(* IEC 61131-3 sources: elnaProjects/ElpcLogic/PomarKc7Changed/FunctionBlocks (part 8) *)

(* ---- Pusk_second_faza_chastotny.st ---- *)
FUNCTION_BLOCK Pusk_second_faza_chastotny

VAR_IN_OUT
	StrAlg : struct_Alg;
END_VAR

VAR
	timer120 : struct_PhaseAlgoritm;
	timer5 : struct_PhaseAlgoritm;
	Shup : struct_PhaseAlgoritm;
	Net_Chast : struct_PhaseAlgoritm;
	mvOn : struct_PhaseAlgoritm;
	pGNSmore04 : struct_PhaseAlgoritm;
	gotov_K_zagruzke : struct_PhaseAlgoritm;
	dPmg_Top : struct_PhaseAlgoritm;
	AutoPNS_Start : struct_PhaseAlgoritm;
	fb_timer120 : fb_ph_Timer;
	fb_timer5 : fb_ph_Timer;
	fb_Shup : fb_ph_OilPump;
	fb_Net_Chast : fb_ph_algoritm;
	fb_mvOn : fb_ph_SectionSwitch;
	fb_pGNSmore04 : fb_ph_algoritm;
	fb_gotov_K_zagruzke : fb_ph_algoritm;
	fb_dPmg_Top : fb_ph_algoritm;
	fb_AutoPNS_Start : fb_ph_algoritm;
	_sunpackerCommand : fb_sunpackerCommand;
	_statusDualInput : TYPE_statusDualInput;
	_Answers : TYPE_Answers;
	source : BYTE;
	cmd : BYTE;
	lastCmd : BYTE;
	source_for_Status : BYTE;
	cmd_for_Status : BYTE;
	command_error_for_Status : BYTE;
	resetCmdTimer : TON;
	resetCmdTimerPriznak : BOOL;
	onInit : BOOL;
	waitReset : TON;
END_VAR

VAR_EXTERNAL
	ModeGpa : TYPE_ModeGpa;
	algManager : struct_AlgoritmsManager;
	IM : ImConfig;
	protections : ProtectionsConfig;
	algoritms : AlgoritmsConfig;
	ai : AiConfig;
END_VAR

VAR
	statusAi : TYPE_StatusAi;
END_VAR

IF NOT onInit THEN
         fb_timer120(phaseNumber:=1, delay:=T#120S);
         fb_timer5(phaseNumber:=2, delay:=T#5S);
         fb_Shup(phaseNumber:=3);
         fb_Net_Chast(phaseNumber:=4);
         fb_mvOn(phaseNumber:=5,  act:=_on);
         fb_pGNSmore04(phaseNumber:=6);
         fb_gotov_K_zagruzke(phaseNumber:=7);
         fb_dPmg_Top(phaseNumber:=8);
         fb_AutoPNS_Start(phaseNumber:=9, act:=_run, waitCompletion:=FALSE);
onInit:=TRUE;
END_IF;

fb_timer120(StrPh:=timer120);
fb_timer5(StrPh:= timer5);
fb_Shup(StrPh:= Shup);
fb_Net_Chast(StrPh:=Net_Chast);
fb_mvOn(StrPh:=mvOn, Im:=IM.mv);
fb_pGNSmore04(StrPh:=pGNSmore04);
fb_gotov_K_zagruzke(StrPh:=gotov_K_zagruzke);
fb_dPmg_Top(StrPh:=dPmg_Top);
fb_AutoPNS_Start(StrPh:=AutoPNS_Start, alg:=algoritms.autoPns);

StrAlg.CanRun := StrAlg.inCanRun;
StrAlg.OpcCommandsDisabled := StrAlg.inOpcCommandsDisabled;

IF StrAlg.isRuning THEN
    (* мв не включен - запуск таймера *)
    IF NOT mvOn.top THEN
	runphase(timer120);
    END_IF;
    (* частотный пуск не совершен - запуск таймера *)
    IF NOT Net_Chast.top THEN
	runphase(timer5);
    END_IF;

    (* ШУП не запущен - запуск *)
    IF NOT Shup.start THEN
	runphase(Shup);
    END_IF;

    (* ШУП не завершился - запуск ШУПб МВ *)
    IF NOT Shup.top AND Shup.start THEN
	runIfNotRunningSO(IM.SingleOutputs.Pusk_SHUP);
	Shup.top:=TRUE;
	runphase(mvOn);
    END_IF;

    (* частотный пуск не запущен - запуск *)
    IF NOT Net_Chast.start THEN
	runphase(Net_Chast);
    END_IF;

    (* частотный пуск не завершился - запуск *)
    IF Net_Chast.start AND (NOT Net_Chast.top) THEN
	IF (NOT IM.SingleSignals.Chastotny_pusk.Q) AND (IM.SingleSignals.Chastotny_pusk.status = 1) THEN
		Net_Chast.top:=TRUE;
		resetPhase(timer5);
	END_IF;
    END_IF;

    (* таймер не истек и мв не включен - вовзедение защиты *)
    IF (NOT timer120.top) AND (NOT mvOn.top) THEN
	runDiProtection(protections.Fail_chastotnii_pusk);
    ELSE
	resetDiProtection(protections.Fail_chastotnii_pusk);
    END_IF;

    (* мв не завершился - включение мв *)
    IF mvOn.start AND NOT mvOn.top THEN
	IF IM.mv.onStatus = _statusDualInput.STATUS_ON THEN
              mvOn.top:=TRUE;
	END_IF;
    END_IF;

    (* мв завершился - что-то делаем *)
    IF mvOn.top THEN
	IF NOT pGNSmore04.start (*AND (algManager.mode = ModeGpa.MODE_PUSKPP_Ch OR algManager.mode = ModeGpa.MODE_PUSKAP_Ch)какой режим *) THEN
		runphase(pGNSmore04);
	END_IF;
         (* IF NOT autoAVOM_canrun_flag THEN
              algoritms.AutoAvom.CanRun:=TRUE;
	    autoAVOM_canrun_flag:=TRUE; kto ti
	END_IF;*)
	resetPhase(timer120);
	runphase(gotov_K_zagruzke);

          IF NOT dPmg_Top.start (* AND ((algManager.mode = modegpa.MODE_PUSKAP_Ch) OR (algManager.mode = modegpa.MODE_PUSKPP_Ch))*) THEN
              runphase(dPmg_Top);
	END_IF;

          runAiProtection(protections.Pgaza_na_vyhode_nagnetatelia_GPA_STOP);
	runDiProtection(protections.Off_avar_vikluchatel);
	runDiProtection(protections.Reg_vozb_off);
    END_IF;

    IF dPmg_Top.start AND NOT dPmg_Top.top THEN
	IF NOT IM.SingleSignals.dP_maslo_gaz_Less100.Q AND IM.SingleSignals.dP_maslo_gaz_Less100.status = 1 AND ai.dPmaslo_gaz.value > 150.0 THEN
		dPmg_Top.top:=TRUE;
		runAiProtection(protections.dPmaslo_gaz);
		runDiProtection(protections.dPmaslo_gaz_less100);
		resetAiProtection(protections.Pgaza_na_vhode_nagnetatelia_GPA_STOP);
		resetAiProtection(protections.Pgaza_na_vyhode_nagnetatelia_GPA_STOP);
		algoritms.autoNu.CanRun:=TRUE;
		(*algoritms.autoNu.run(); кого чего, ничего не понимаю *)
	END_IF;
    END_IF;

    IF pGNSmore04.start AND NOT pGNSmore04.top THEN
	IF ai.Pmasla_posle_GNS.interval (*почему интервал, если есть статус *) >= statusAi.NORMAL AND ai.Pmasla_posle_GNS.value > 400.0 THEN
	  	pGNSmore04.top:=TRUE;
	END_IF;
    END_IF;

    IF (pGNSmore04.top AND gotov_K_zagruzke.top AND dPmg_Top.top )(*AND (algManager.mode = modegpa.MODE_PUSKAP_Ch OR (algManager.mode = modegpa.MODE_PUSKPP_Ch) *)OR
	(gotov_K_zagruzke.top) (*AND (algManager.mode = modegpa.MODE_PUSKV_Ch OR algManager.mode = modegpa.MODE_I))*) AND NOT AutoPNS_Start.top  THEN
	algoritms.AutoPns.CanRun :=TRUE;
	(*algoritms.AutoPns;*)
	AutoPNS_Start.top:=TRUE;
    END_IF;

    IF (NOT Net_Chast.top AND timer5.top) OR (timer120.top AND NOT mvOn.top) THEN
	algoritms.ao.CanRun:=TRUE;
	(*algoritms.ao.run ();*)
    END_IF;
END_IF;

StrAlg.CanRun := StrAlg.inCanRun;
StrAlg.OpcCommandsDisabled := StrAlg.inOpcCommandsDisabled;

(* ---- Если управление с ВУ заблокировано, то  передаем команду из алгоритма ---- *)
IF StrAlg.inOpcCommandsDisabled THEN
	StrAlg.inCommand := StrAlg.inCommand_Alg;
ELSE (* иначе передаем команду с АРМа*)
	StrAlg.inCommand := StrAlg.inCommand_ARM;
END_IF;

_sunpackerCommand(command := StrAlg.inCommand);
	source := _sunpackerCommand.source;
	cmd := _sunpackerCommand.cmd;

IF cmd <> 0 AND lastCmd <> cmd AND (((NOT StrAlg.opcCommandsDisabled) AND source > 0) OR source = 0) then
	CASE BYTE_TO_INT(cmd) OF
		(*cmdRun*) 1: 	IF (StrAlg.CanRun) THEN
					StrAlg.isRuning := TRUE;
					StrAlg.isEnded := FALSE;
					StrAlg.hasError := FALSE;
					(*****************       OnRun       *****************)
                                                  algManager.nMode:=ModeGpa.MODE_PUSK_FIRST_FAZA2;

                                                  runPhase(timer120);
                                                  runPhase(timer5);
                                                  runPhase(Shup);
                                                  resetAiProtection(protections.dPmaslo_gaz);
                                                  resetDiProtection(protections.dPmaslo_gaz_less100);

					cmd_for_Status := cmd;
					source_for_Status := source;
					command_error_for_Status := 0;
				ELSE
					StrAlg.isRuning := FALSE;
					StrAlg.isEnded := FALSE;
					StrAlg.hasError := FALSE;

					cmd_for_Status := 0;
					source_for_Status := source;
					command_error_for_Status := cmd;
				END_IF;
		(*cmdReset*) 2: 	StrAlg.isRuning := FALSE;
				StrAlg.isEnded := FALSE;
				StrAlg.hasError 	:= FALSE;

                                         (*****************       OnReset       *****************)
                                        waitReset(IN:=FALSE);
                                        StrAlg.inCanRun:=FALSE;

                                        resetPhase(timer5);
                                        resetPhase(Shup);
                                        resetPhase(timer120);
                                        resetPhase(Net_Chast);
                                        resetPhase(mvOn);
                                        resetPhase(pGNSmore04);
                                        resetPhase(gotov_K_zagruzke);
                                        resetPhase(dPmg_Top);
                                        resetPhase(AutoPNS_Start);

                                        StrAlg.inOpcCommandsDisabled:=FALSE;

				cmd_for_Status := cmd;
				source_for_Status := source;
				command_error_for_Status := 0;
	END_CASE;
	resetCmdTimer(IN := false);
	resetCmdTimerPriznak := TRUE;
END_IF;
lastCmd := cmd;

resetCmdTimer(IN := resetCmdTimerPriznak, PT := T#5S);
IF resetCmdTimer.Q THEN
	resetCmdTimerPriznak := FALSE;
	source_for_Status := 0;
	cmd_for_Status := 0;
	command_error_for_Status := 0;
END_IF;

StrAlg.Start:= timer120.startStatus
            OR timer5.startStatus
            OR Shup.startStatus
            OR Net_Chast.startStatus
            OR mvOn.startStatus
            OR pGNSmore04.startStatus
            OR gotov_K_zagruzke.startStatus
            OR dPmg_Top.startStatus
            OR AutoPNS_Start.startStatus;

StrAlg.Error := timer120.errorStatus
            OR timer5.errorStatus
            OR Shup.errorStatus
            OR Net_Chast.errorStatus
            OR mvOn.errorStatus
            OR pGNSmore04.errorStatus
            OR gotov_K_zagruzke.errorStatus
            OR dPmg_Top.errorStatus
            OR AutoPNS_Start.errorStatus;

StrAlg.Top := timer120.topStatus
            OR timer5.topStatus
            OR Shup.topStatus
            OR Net_Chast.topStatus
            OR mvOn.topStatus
            OR gotov_K_zagruzke.topStatus
            OR dPmg_Top.topStatus
            OR AutoPNS_Start.topStatus
            OR pGNSmore04.topStatus;

(*TODO: TYPE PROGRAM CODE HERE*)
StrAlg.status :=  SHL(BYTE_TO_DWORD(source_for_Status), 29)
			OR SHL(BYTE_TO_DWORD(cmd_for_Status), 26)
			OR SHL(BYTE_TO_DWORD(command_error_for_Status), 23)
			OR SHL(BOOL_TO_DWORD(StrAlg.OpcCommandsDisabled ), 21)
			OR SHL(BOOL_TO_DWORD(StrAlg.hasError),4)
			OR SHL(BOOL_TO_DWORD(StrAlg.CanRun),2)
			OR SHL(BOOL_TO_DWORD(StrAlg.isEnded),1)
			OR BOOL_TO_DWORD(StrAlg.isRuning);

(* ---- Pusk_second_faza_reactor.st ---- *)
FUNCTION_BLOCK Pusk_second_faza_reactor

VAR_IN_OUT
	StrAlg : struct_Alg;
END_VAR

VAR
	timer25 : struct_PhaseAlgoritm;
	timer3 : struct_PhaseAlgoritm;
	mvOn : struct_PhaseAlgoritm;
	pGNSmore04 : struct_PhaseAlgoritm;
	gotov_K_zagruzke : struct_PhaseAlgoritm;
	dPmg_Top : struct_PhaseAlgoritm;
	Mv_Error : struct_PhaseAlgoritm;
	AutoPNS_Start : struct_PhaseAlgoritm;
	fb_timer25 : fb_ph_Timer;
	fb_timer3 : fb_ph_Timer;
	fb_Mv_Error : fb_ph_algoritm;
	fb_mvOn : fb_ph_SectionSwitch;
	fb_pGNSmore04 : fb_ph_algoritm;
	fb_gotov_K_zagruzke : fb_ph_algoritm;
	fb_dPmg_Top : fb_ph_algoritm;
	fb_AutoPNS_Start : fb_ph_algoritm;
	_sunpackerCommand : fb_sunpackerCommand;
	_statusDualInput : TYPE_statusDualInput;
	_Answers : TYPE_Answers;
	source : BYTE;
	cmd : BYTE;
	lastCmd : BYTE;
	source_for_Status : BYTE;
	cmd_for_Status : BYTE;
	command_error_for_Status : BYTE;
	resetCmdTimer : TON;
	resetCmdTimerPriznak : BOOL;
	onInit : BOOL;
	waitReset : TON;
END_VAR

VAR_EXTERNAL
	ModeGpa : TYPE_ModeGpa;
	algManager : struct_AlgoritmsManager;
	IM : ImConfig;
	protections : ProtectionsConfig;
	algoritms : AlgoritmsConfig;
	ai : AiConfig;
END_VAR

VAR
	statusAi : TYPE_StatusAi;
END_VAR

IF NOT onInit THEN
         fb_timer25(phaseNumber:=1, delay:=T#25S);
         fb_timer3(phaseNumber:=2, delay:=T#3S);
         fb_mvOn(phaseNumber:=3, act:=_on);
         fb_pGNSmore04(phaseNumber:=4);
         fb_gotov_K_zagruzke(phaseNumber:=5);
         fb_dPmg_Top(phaseNumber:=6);
         fb_Mv_Error(phaseNumber:=7);
         fb_AutoPNS_start(phaseNumber:=8, act:=_run, waitCompletion:=FALSE);

onInit:=TRUE;
END_IF;

fb_timer25(StrPh:=timer25);
fb_timer3(StrPh:= timer3);
fb_mvOn(StrPh:= mvOn, Im:=IM.mv);
fb_pGNSmore04(StrPh:=pGNSmore04);
fb_gotov_K_zagruzke(StrPh:=gotov_K_zagruzke);
fb_dPmg_Top(StrPh:=dPmg_Top);
fb_Mv_Error(StrPh:=Mv_Error);
fb_AutoPNS_start(StrPh:=AutoPNS_start, alg:=algoritms.autoPns);

StrAlg.CanRun := StrAlg.inCanRun;
StrAlg.OpcCommandsDisabled := StrAlg.inOpcCommandsDisabled;
IF StrAlg.isRuning THEN
    (* если мв не завершен - включаем таймер *)
    IF NOT mvOn.top THEN
        runPhase(timer25);
    END_IF;

    (* если мв не заврешен - включаем таймер *)
    IF NOT mvOn.top THEN
        runPhase(timer3);
    END_IF;

    (* мв не запущен - запускаем мв *)
    IF NOT mvOn.start THEN
        runPhase(mvOn);
    END_IF;

    (* мв завершен *)
    IF mvOn.top  THEN
    (*если проверка пгнс не включена - включаем *)
        IF NOT pGNSmore04.start (*AND ((algManager.mode = modegpa.MODE_PUSKAP_R) OR (algManager.mode = modegpa.MODE_PUSKPP_R))*) THEN
            runPhase(pGNSmore04);
        END_IF;

        (*kakoito flag, hz zachem on
        IF NOT autoAVOM_canrun_flag THEN
            algoritms.S_AutoAVOM.CanRun:=TRUE;
            autoAVOM_canrun_flag:=TRUE;
        END_IF;*)
        resetPhase(timer3);
        resetPhase(timer25);
        Mv_Error.error := FALSE;
        runPhase(gotov_K_zagruzke);
        IF NOT dPmg_Top.start (*AND ((algManager.mode = modegpa.MODE_PUSKAP_R) OR (algManager.mode = modegpa.MODE_PUSKPP_R))*) THEN
            runPhase(dPmg_Top);
        END_IF;

        runDiProtection(protections.mvOff);
        runDiProtection(protections.Off_avar_vikluchatel);
        runDiProtection(protections.Reg_vozb_off);
        ELSIF NOT mvOn.top AND timer3.top THEN
		Mv_Error.error := TRUE;
    END_IF;

    IF	dPmg_Top.start AND NOT dPmg_Top.top THEN
	    IF	NOT IM.SingleSignals.dP_maslo_gaz_Less100.Q AND IM.SingleSignals.dP_maslo_gaz_Less100.status = 1 AND ai.dPmaslo_gaz.value > 150.0	THEN
		    dPmg_Top.top:=TRUE;
		    runAiProtection(protections.dPmaslo_gaz);
		    runDiProtection(protections.dPmaslo_gaz_less100);
		    resetAiProtection(protections.Pgaza_na_vhode_nagnetatelia_GPA_STOP);
		    resetAiProtection(protections.Pgaza_na_vyhode_nagnetatelia_GPA_STOP);
		    (*algoritms.autoNu_2.CanRun:=TRUE;
		    algoritms.autoNu_2.run (); не понимаю*)
	    END_IF;
    END_IF;

    IF	pGNSmore04.start AND NOT pGNSmore04.top THEN
	    IF 	ai.Pmasla_posle_GNS.interval	>=statusAi.NORMAL AND ai.Pmasla_posle_GNS.value	 > 400.0 THEN
	  	    pGNSmore04.top:=TRUE;
	    END_IF;
    END_IF;

    IF	pGNSmore04.top AND gotov_K_zagruzke.top AND dPmg_Top.top (*AND algManager.mode = modegpa.MODE_PUSKAP_R) OR (algManager.mode = modegpa.MODE_PUSKPP_R)))*) OR
	    gotov_K_zagruzke.top (*AND ((algManager.mode = modegpa.MODE_PUSKV_R) OR (algManager.mode = modegpa.MODE_I))))*) AND NOT AutoPNS_start.top  THEN
	    algoritms.AutoPns.CanRun :=TRUE;
	   (*algoritms.AutoPNS_Start.run();*)
	    AutoPNS_start.top:=TRUE;
    END_IF;
    IF	timer25.top AND Mv_Error.error THEN
	algoritms.ao.CanRun:=TRUE;
	(*algoritms.ao.run ();*)
    END_IF;

    (*StrAlg.isEnded:= avom1cmdOff.top AND avom2cmdOff.top;*)
END_IF;
StrAlg.CanRun := StrAlg.inCanRun;
StrAlg.OpcCommandsDisabled := StrAlg.inOpcCommandsDisabled;

(* ---- Если управление с ВУ заблокировано, то  передаем команду из алгоритма ---- *)
IF StrAlg.inOpcCommandsDisabled THEN
	StrAlg.inCommand := StrAlg.inCommand_Alg;
ELSE (* иначе передаем команду с АРМа*)
	StrAlg.inCommand := StrAlg.inCommand_ARM;
END_IF;

_sunpackerCommand(command := StrAlg.inCommand);
	source := _sunpackerCommand.source;
	cmd := _sunpackerCommand.cmd;

IF cmd <> 0 AND lastCmd <> cmd AND (((NOT StrAlg.opcCommandsDisabled) AND source > 0) OR source = 0) then
	CASE BYTE_TO_INT(cmd) OF
		(*cmdRun*) 1: 	IF (StrAlg.CanRun) THEN
					StrAlg.isRuning := TRUE;
					StrAlg.isEnded := FALSE;
					StrAlg.hasError := FALSE;
					(*****************       OnRun       *****************)
                                                  algManager.nMode:=ModeGpa.MODE_PUSK_FIRST_FAZA2;

                                                  (*runPhase(timer120);
                                                  runPhase(timer5);
                                                  runPhase(Shup);
                                                  resetAiProtection(protections.dPmaslo_gaz);
                                                  resetDiProtection(protections.dPmaslo_gaz_less100);*)

					cmd_for_Status := cmd;
					source_for_Status := source;
					command_error_for_Status := 0;
				ELSE
					StrAlg.isRuning := FALSE;
					StrAlg.isEnded := FALSE;
					StrAlg.hasError := FALSE;

					cmd_for_Status := 0;
					source_for_Status := source;
					command_error_for_Status := cmd;
				END_IF;
		(*cmdReset*) 2: 	StrAlg.isRuning := FALSE;
				StrAlg.isEnded := FALSE;
				StrAlg.hasError 	:= FALSE;

                                         (*****************       OnReset       *****************)
                                        waitReset(IN:=FALSE);
                                        StrAlg.inCanRun:=FALSE;

                                        (*resetPhase(timer5);
                                        resetPhase(Shup);
                                        resetPhase(timer120);
                                        resetPhase(Net_Chast);
                                        resetPhase(mvOn);
                                        resetPhase(pGNSmore04);
                                        resetPhase(gotov_K_zagruzke);
                                        resetPhase(dPmg_Top);
                                        resetPhase(AutoPNS_Start);*)

                                        StrAlg.inOpcCommandsDisabled:=FALSE;

				cmd_for_Status := cmd;
				source_for_Status := source;
				command_error_for_Status := 0;
	END_CASE;
	resetCmdTimer(IN := false);
	resetCmdTimerPriznak := TRUE;
END_IF;
lastCmd := cmd;

resetCmdTimer(IN := resetCmdTimerPriznak, PT := T#5S);
IF resetCmdTimer.Q THEN
	resetCmdTimerPriznak := FALSE;
	source_for_Status := 0;
	cmd_for_Status := 0;
	command_error_for_Status := 0;
END_IF;

StrAlg.Start:= timer25.errorStatus
            OR timer3.errorStatus
            OR mvOn.errorStatus
            OR pGNSmore04.errorStatus
            OR gotov_K_zagruzke.errorStatus
            OR dPmg_Top.errorStatus
            OR Mv_Error.errorStatus
            OR AutoPNS_Start.errorStatus;

(*TODO: TYPE PROGRAM CODE HERE*)
StrAlg.status :=  SHL(BYTE_TO_DWORD(source_for_Status), 29)
			OR SHL(BYTE_TO_DWORD(cmd_for_Status), 26)
			OR SHL(BYTE_TO_DWORD(command_error_for_Status), 23)
			OR SHL(BOOL_TO_DWORD(StrAlg.OpcCommandsDisabled ), 21)
			OR SHL(BOOL_TO_DWORD(StrAlg.hasError),4)
			OR SHL(BOOL_TO_DWORD(StrAlg.CanRun),2)
			OR SHL(BOOL_TO_DWORD(StrAlg.isEnded),1)
			OR BOOL_TO_DWORD(StrAlg.isRuning);

(* ---- Pusk_third_faza.st ---- *)
FUNCTION_BLOCK Pusk_third_faza

VAR_IN_OUT
	StrAlg : struct_Alg;
END_VAR

VAR
	timer480 : struct_PhaseAlgoritm;
	kran4Open : struct_PhaseAlgoritm;
	waitAfterKran4 : struct_PhaseAlgoritm;
	kran5Close : struct_PhaseAlgoritm;
	kran3bOpen : struct_PhaseAlgoritm;
	dP_kr1less100 : struct_PhaseAlgoritm;
	Pvh_vyhMore5 : struct_PhaseAlgoritm;
	kran1Open : struct_PhaseAlgoritm;
	kran2Open : struct_PhaseAlgoritm;
	kran3Open : struct_PhaseAlgoritm;
	kran3bClose : struct_PhaseAlgoritm;
	Err_ALG : struct_PhaseAlgoritm;
	fb_timer480 : fb_ph_Timer;
	fb_kran4Open : fb_ph_Kran;
	fb_waitAfterKran4 : fb_ph_Timer;
	fb_kran5Close : fb_ph_Kran;
	fb_kran3bOpen : fb_ph_Kran;
	fb_dP_kr1less100 : fb_ph_algoritm;
	fb_Pvh_vyhMore5 : fb_ph_algoritm;
	fb_kran1Open : fb_ph_Kran;
	fb_kran2Open : fb_ph_Kran;
	fb_kran3Open : fb_ph_Kran;
	fb_kran3bClose : fb_ph_Kran;
	fb_Err_ALG : fb_ph_algoritm;
	_sunpackerCommand : fb_sunpackerCommand;
	_statusDualInput : TYPE_statusDualInput;
	_Answers : TYPE_Answers;
	source : BYTE;
	cmd : BYTE;
	lastCmd : BYTE;
	source_for_Status : BYTE;
	cmd_for_Status : BYTE;
	command_error_for_Status : BYTE;
	resetCmdTimer : TON;
	resetCmdTimerPriznak : BOOL;
	onInit : BOOL;
	waitReset : TON;
END_VAR

VAR_EXTERNAL
	ModeGpa : TYPE_ModeGpa;
	algManager : struct_AlgoritmsManager;
	IM : ImConfig;
	protections : ProtectionsConfig;
	algoritms : AlgoritmsConfig;
	ai : AiConfig;
END_VAR

VAR
	statusAi : TYPE_StatusAi;
END_VAR

IF NOT onInit THEN
         fb_timer480(phaseNumber:=1, delay:=T#480S);
         fb_kran4Open(phaseNumber:=2, act:=_on);
         fb_waitAfterKran4(phaseNumber:=3, delay:=T#10S);
         fb_kran5Close(phaseNumber:=4, act:=_off);
         fb_kran3bOpen(phaseNumber:=5, act:=_on);
         fb_dP_kr1less100(phaseNumber:=6);
         fb_Pvh_vyhMore5(phaseNumber:=7);
         fb_kran1Open(phaseNumber:=8, act:=_on);
         fb_kran2Open(phaseNumber:=9, act:=_on);
         fb_kran3Open(phaseNumber:=10, act:=_on);
         fb_kran3bClose(phaseNumber:=11, act:=_off);
         fb_Err_ALG(phaseNumber:=12);
onInit:=TRUE;
END_IF;

fb_timer480(StrPh:=timer480);
fb_kran4Open(StrPh:= kran4Open, Im:=Im.kran4);
fb_waitAfterKran4(StrPh:= waitAfterKran4);
fb_kran5Close(StrPh:=kran5Close, Im:=Im.kran5);
fb_kran3bOpen(StrPh:=kran3bOpen, Im:=Im.kran3b);
fb_dP_kr1less100(StrPh:=dP_kr1less100);
fb_Pvh_vyhMore5(StrPh:=Pvh_vyhMore5);
fb_kran1Open(StrPh:=kran1Open, Im:=Im.kran1);
fb_kran2Open(StrPh:=kran2Open, Im:=Im.kran2);
fb_kran3Open(StrPh:=kran3Open, Im:=Im.kran3);
fb_kran3bClose(StrPh:=kran3bClose, Im:=Im.kran3b);
fb_Err_ALG(StrPh:=Err_ALG);

StrAlg.CanRun := StrAlg.inCanRun;
StrAlg.OpcCommandsDisabled := StrAlg.inOpcCommandsDisabled;

IF StrAlg.isRuning THEN
    (* запуск таймера *)
    IF NOT (kran3bClose.top) THEN
	    runPhase(timer480);
    END_IF;

    (*если кран1 не открыт - октрыть кран 4*)
    IF	NOT kran1Open.top (*AND IM.kran4._cmdreset.IN = FALSE*)  THEN
	    runIfNotRunningSO(IM.SingleOutputs.Kr4_open_from_alg);
	    runPhase(kran4Open);
    END_IF;
    IF	kran4Open.start AND NOT kran4Open.top THEN
	    IF	IM.kran4.onStatus = _statusDualInput.STATUS_ON THEN
		    kran4Open.top:=TRUE;
	    END_IF;
    END_IF;

    (* продувка крана *)
    IF kran4Open.top THEN
        runPhase(waitAfterKran4);
    END_IF;

    (* кран продулся - закрытие кран 5*)
    IF waitAfterKran4.top THEN
	    runPhase(kran5Close);
    END_IF;

    (* кран 5 закрыт - открытие крана 3б проверка перепада давление*)
    IF	kran5Close.top THEN
	    runPhase(kran3bOpen);
	    runPhase(dP_kr1less100);
	    runPhase(Pvh_vyhMore5);
    END_IF;

    (* проверка давления крана *)
    IF	Pvh_vyhMore5.start AND NOT Pvh_vyhMore5.top THEN
	    IF	(ai.Pgaza_na_vhode_nagnetatelia.interval >=statusAi.NORMAL) AND (ai.Pgaza_na_vhode_nagnetatelia.value	 >= 4.0) AND
		    (ai.Pgaza_na_vyhode_nagnetatelia.interval >=statusAi.NORMAL) AND (ai.Pgaza_na_vyhode_nagnetatelia.value	 >= 4.0) THEN
		        Pvh_vyhMore5.top := TRUE;
    		    runAiProtection(protections.Pgaza_na_vyhode_nagnetatelia);
	    END_IF;
    END_IF;

    (* проверка открытия крана 3б *)
    IF	kran3bOpen.start AND NOT kran3bOpen.top THEN
	    IF	IM.kran3b.onStatus=_statusDualInput.STATUS_ON THEN
		    kran3bOpen.top :=TRUE;
	    END_IF;
    END_IF;
    IF	kran3bOpen.top AND	kran5Close.top AND dP_kr1less100.top AND Pvh_vyhMore5.top THEN
	    runPhase(kran1Open);
	    runPhase(kran2Open);
	    runPhase(kran3Open);
	    (*Smazka_1_2:=TRUE; нет такого *)
    END_IF;
    IF	kran1Open.top THEN
	    resetIfRunningSO(IM.SingleOutputs.Kr4_open_from_alg);
	    (*ystavki.Block_kr4_alg.setValue (0);что такое уставки*)
    END_IF;

    (* закрытие крана 3бис *)
    IF kran1Open.top AND kran2Open.top AND kran3Open.top THEN
	    runPhase(kran3bClose);
    END_IF;
    IF 	kran3bClose.top THEN
	    Err_ALG.error :=FALSE;
	    resetPhase(timer480);
    ELSIF NOT kran3bClose.top AND timer480.top THEN
		Err_ALG.error :=TRUE;
    END_IF;
END_IF;

_sunpackerCommand(command := StrAlg.inCommand);
	source := _sunpackerCommand.source;
	cmd := _sunpackerCommand.cmd;

IF cmd <> 0 AND lastCmd <> cmd AND (((NOT StrAlg.opcCommandsDisabled) AND source > 0) OR source = 0) then
	CASE BYTE_TO_INT(cmd) OF
		(*cmdRun*) 1: 	IF (StrAlg.CanRun) THEN
					StrAlg.isRuning := TRUE;
					StrAlg.isEnded := FALSE;
					StrAlg.hasError := FALSE;
					(*****************       OnRun       *****************)
                                                  algManager.nMode:=ModeGpa.MODE_PUSK_FIRST_FAZA2;

                                                  (*runPhase(timer120);
                                                  runPhase(timer5);
                                                  runPhase(Shup);
                                                  resetAiProtection(protections.dPmaslo_gaz);
                                                  resetDiProtection(protections.dPmaslo_gaz_less100);*)

					cmd_for_Status := cmd;
					source_for_Status := source;
					command_error_for_Status := 0;
				ELSE
					StrAlg.isRuning := FALSE;
					StrAlg.isEnded := FALSE;
					StrAlg.hasError := FALSE;

					cmd_for_Status := 0;
					source_for_Status := source;
					command_error_for_Status := cmd;
				END_IF;
		(*cmdReset*) 2: 	StrAlg.isRuning := FALSE;
				StrAlg.isEnded := FALSE;
				StrAlg.hasError 	:= FALSE;

                                         (*****************       OnReset       *****************)
                                        waitReset(IN:=FALSE);
                                        StrAlg.inCanRun:=FALSE;

                                        (*resetPhase(timer5);
                                        resetPhase(Shup);
                                        resetPhase(timer120);
                                        resetPhase(Net_Chast);
                                        resetPhase(mvOn);
                                        resetPhase(pGNSmore04);
                                        resetPhase(gotov_K_zagruzke);
                                        resetPhase(dPmg_Top);
                                        resetPhase(AutoPNS_Start);*)

                                        StrAlg.inOpcCommandsDisabled:=FALSE;

				cmd_for_Status := cmd;
				source_for_Status := source;
				command_error_for_Status := 0;
	END_CASE;
	resetCmdTimer(IN := false);
	resetCmdTimerPriznak := TRUE;
END_IF;
lastCmd := cmd;

resetCmdTimer(IN := resetCmdTimerPriznak, PT := T#5S);
IF resetCmdTimer.Q THEN
	resetCmdTimerPriznak := FALSE;
	source_for_Status := 0;
	cmd_for_Status := 0;
	command_error_for_Status := 0;
END_IF;

StrAlg.Start:= timer480.startStatus
            OR kran4Open.startStatus
            OR waitAfterKran4.startStatus
            OR kran5Close.startStatus
            OR kran3bOpen.startStatus
            OR dP_kr1less100.startStatus
            OR Pvh_vyhMore5.startStatus
            OR kran1Open.startStatus
            OR kran2Open.startStatus
            OR kran3Open.startStatus
            OR kran3bClose.startStatus
            OR Err_ALG.startStatus;

StrAlg.Error := timer480.errorStatus
            OR kran4Open.errorStatus
            OR waitAfterKran4.errorStatus
            OR kran5Close.errorStatus
            OR kran3bOpen.errorStatus
            OR dP_kr1less100.errorStatus
            OR Pvh_vyhMore5.errorStatus
            OR kran1Open.errorStatus
            OR kran2Open.errorStatus
            OR kran3Open.errorStatus
            OR kran3bClose.errorStatus
            OR Err_ALG.errorStatus;

StrAlg.Top := timer480.topStatus
            OR kran4Open.topStatus
            OR waitAfterKran4.topStatus
            OR kran5Close.topStatus
            OR kran3bOpen.topStatus
            OR dP_kr1less100.topStatus
            OR Pvh_vyhMore5.topStatus
            OR kran1Open.topStatus
            OR kran2Open.topStatus
            OR kran3Open.topStatus
            OR kran3bClose.topStatus
            OR Err_ALG.topStatus;

(*TODO: TYPE PROGRAM CODE HERE*)
StrAlg.status :=  SHL(BYTE_TO_DWORD(source_for_Status), 29)
			OR SHL(BYTE_TO_DWORD(cmd_for_Status), 26)
			OR SHL(BYTE_TO_DWORD(command_error_for_Status), 23)
			OR SHL(BOOL_TO_DWORD(StrAlg.OpcCommandsDisabled ), 21)
			OR SHL(BOOL_TO_DWORD(StrAlg.hasError),4)
			OR SHL(BOOL_TO_DWORD(StrAlg.CanRun),2)
			OR SHL(BOOL_TO_DWORD(StrAlg.isEnded),1)
			OR BOOL_TO_DWORD(StrAlg.isRuning);

(* ---- puskKalg.st ---- *)
FUNCTION_BLOCK puskKalg

VAR_IN_OUT
	StrAlg : struct_Alg;
END_VAR

VAR
	puskOilSystem : struct_PhaseAlgoritm;
END_VAR

VAR_IN_OUT
	questionFilling : struct_Question;
END_VAR

VAR
	filling : struct_PhaseAlgoritm;
END_VAR

VAR_IN_OUT
	questionUnload : struct_Question;
END_VAR

VAR
	kran3bOpen : struct_PhaseAlgoritm;
	kran4Close : struct_PhaseAlgoritm;
	kran1Close : struct_PhaseAlgoritm;
	kran2Close : struct_PhaseAlgoritm;
	kran5open : struct_PhaseAlgoritm;
	wait720 : struct_PhaseAlgoritm;
	noGasInPipe : struct_PhaseAlgoritm;
	AutoNUoff : struct_PhaseAlgoritm;
	nu1Off : struct_PhaseAlgoritm;
	nu2Off : struct_PhaseAlgoritm;
	pnsWaitOff : struct_PhaseAlgoritm;
	testUnsuccessfulUnfill : struct_PhaseAlgoritm;
	fb_puskOilSystem : fb_ph_algoritm;
	fb_questionFilling : fb_Question;
	fb_filling : fb_ph_algoritm;
	fb_questionUnload : fb_Question;
	fb_kran3bOpen : fb_ph_Kran;
	fb_kran4Close : fb_ph_CustomPhase;
	fb_kran1Close : fb_ph_Kran;
	fb_kran2Close : fb_ph_Kran;
	fb_kran5open : fb_ph_Kran;
	fb_wait720 : fb_ph_Timer;
	fb_noGasInPipe : fb_ph_CustomPhase;
	fb_AutoNUoff : fb_ph_algoritm;
	fb_nu1Off : fb_ph_OilPump;
	fb_nu2Off : fb_ph_OilPump;
	fb_pnsWaitOff : fb_ph_algoritm;
	fb_testUnsuccessfulUnfill : fb_ph_CustomPhase;
	_sunpackerCommand : fb_sunpackerCommand;
	_DualStateImAction : TYPE_DualStateImAction;
	_Answers : TYPE_Answers;
	_statusDualInput : TYPE_statusDualInput;
	_StatusAi : TYPE_StatusAi;
	_PhaseAlgoritmAction : TYPE_PhaseAlgoritmAction;
	source : BYTE;
	cmd : BYTE;
	lastCmd : BYTE;
	source_for_Status : BYTE;
	cmd_for_Status : BYTE;
	command_error_for_Status : BYTE;
	resetCmdTimer : TON;
	resetCmdTimerPriznak : BOOL;
	OpcCommandsKransEnabled : BOOL;
	OpcCommandsKransDisabled : BOOL;
	_resetQuestion1 : BOOL;
	_resetQuestion2 : BOOL;
	onInit : BOOL;
	waitReset : TON;
END_VAR

VAR_EXTERNAL
	IM : ImConfig;
	algoritms : AlgoritmsConfig;
	ai : AiConfig;
	AlgTimers : struct_AlgTimers;
	ModeGpa : TYPE_ModeGpa;
	algManager : struct_AlgoritmsManager;
	protections : ProtectionsConfig;
END_VAR

VAR CONSTANT
	Ust_Pgaza : LREAL          := 0.3;
END_VAR

IF NOT onInit THEN

          fb_puskOilSystem(phaseNumber:=0, act:=_run, waitCompletion:=TRUE);
      questionFilling.AnswerVariants:=_Answers.ANS_YES;
                fb_filling(phaseNumber:=1, act:=_run, waitCompletion:=TRUE);
    questionUnload.AnswerVariants:=_Answers.ANS_YES;
             fb_kran3bOpen(phaseNumber:=3, act:=_on);
             fb_kran4Close(phaseNumber:=4);
             fb_kran1Close(phaseNumber:=5, act:=_off);
             fb_kran2Close(phaseNumber:=6, act:=_off);
              fb_kran5open(phaseNumber:=7, act:=_on);
                fb_wait720(phaseNumber:=8, delay:=T#720S);
            fb_noGasInPipe(phaseNumber:=9);
              fb_AutoNUoff(phaseNumber:=10, act:=_reset, waitCompletion:=FALSE);
                 fb_nu1Off(phaseNumber:=11, act:=_off);
                 fb_nu2Off(phaseNumber:=12, act:=_off);
             fb_pnsWaitOff(phaseNumber:=15, act:=_run, waitCompletion:=TRUE);
 fb_testUnsuccessfulUnfill(phaseNumber:=18);

onInit:=TRUE;
END_IF;

          fb_puskOilSystem(StrPh:=puskOilSystem, alg:=algoritms.puskOilSystem);
        fb_questionFilling(StrQ:=questionFilling);
                fb_filling(StrPh:=filling, alg:=algoritms.filling);
         fb_questionUnload(StrQ:=questionUnload);
             fb_kran3bOpen(StrPh:=kran3bOpen, Im:=Im.kran3b);
             fb_kran4Close(StrPh:=kran4Close);
             fb_kran1Close(StrPh:=kran1Close, Im:=Im.kran1);
             fb_kran2Close(StrPh:=kran2Close, Im:=Im.kran2);
              fb_kran5open(StrPh:=kran5open, Im:=Im.kran5);
                fb_wait720(StrPh:=wait720, timer:=AlgTimers.puskK_wait720);
            fb_noGasInPipe(StrPh:=noGasInPipe);
              fb_AutoNUoff(StrPh:=AutoNUoff, alg:=algoritms.autoNu);
                 fb_nu1Off(StrPh:=nu1Off, Im:=Im.nu1);
                 fb_nu2Off(StrPh:=nu2Off, Im:=Im.nu2);
             fb_pnsWaitOff(StrPh:=pnsWaitOff, alg:=algoritms.vibegPNS);
 fb_testUnsuccessfulUnfill(StrPh:=testUnsuccessfulUnfill);

StrAlg.CanRun := StrAlg.inCanRun;
StrAlg.OpcCommandsDisabled := StrAlg.inOpcCommandsDisabled;

IF StrAlg.isRuning THEN

    StrAlg.hasError := kran3bOpen.error OR kran1Close.error OR kran2Close.error OR kran5open.error OR testUnsuccessfulUnfill.error;

    IF puskOilSystem.top THEN
         IF NOT _resetQuestion1 THEN
         askQuestion(questionFilling);
         _resetQuestion1:=TRUE;
         END_IF;
    END_IF;

    IF questionFilling.answer = _Answers.ANS_YES THEN
        runPhase(filling);
        resetQuestion(questionFilling);
    END_IF;

    IF filling.top THEN
       OpcCommandsKransEnabled:=TRUE;
       resetDiProtection(protections.Reg_vozb_off);
       (*resetDiProtection(protections.Fail_chastotnii_pusk);*)
       IF NOT _resetQuestion2 THEN
       askQuestion(questionUnload);
       _resetQuestion2:=TRUE;
       END_IF;
    END_IF;

     IF questionUnload.answer = _Answers.ANS_YES THEN
        OpcCommandsKransDisabled:=TRUE;
        runPhase(kran3bOpen);
        runPhase(wait720);
        resetQuestion(questionUnload);
    END_IF;

    IF kran3bOpen.top THEN
          resetDiProtection(protections.Reg_vozb_off);
          resetDiProtection(protections.Fail_chastotnii_pusk);

          runPhase(kran1Close);
          runPhase(kran2Close);
          runPhase(kran4Close);
    END_IF;

     IF kran4Close.start AND NOT kran4Close.top THEN
	kran4Close.top:= Im.kran4.onStatus = _statusDualInput.STATUS_OFF;
    END_IF;

    IF kran1Close.top AND kran2Close.top AND kran4Close.top THEN
	runPhase(kran5open);
    END_IF;

    IF kran5open.top THEN
	runPhase(noGasInPipe);
    END_IF;

    IF noGasInPipe.start AND (NOT noGasInPipe.top) THEN
	noGasInPipe.top:=  (ai.dPgaza_na_maslo_filtre.interval >= _statusAi.NORMAL
                         AND  ai.dPgaza_na_maslo_filtre.value< Ust_Pgaza )
                         AND (ai.Pmaslo_sm_vysokoe.interval >= _statusAi.NORMAL
                         AND  ai.Pmaslo_sm_vysokoe.value< Ust_Pgaza);
    END_IF;

    IF noGasInPipe.top THEN

          ai.Tmasla_MB.Disabled_LA:=TRUE;
          ai.Tmasla_MB.Disabled_LW:=TRUE;
          (*IM.SingleSignals.dP_oilgaz_low.Disabled_Sig:=TRUE;*)
          resetAiProtection(protections.Os_sdvig_nagnetatelja_plus);
         (* resetDiProtection(protections.Vibro_skorost_OP_shesterni_RED_T5);*)
	runPhase(AutoNUoff);

    END_IF;

     IF autoNuOff.top THEN
	runPhase(nu1off);
          runPhase(nu2off);
    END_IF;

    IF nu1Off.top AND nu2Off.top THEN
	runPhase(pnsWaitOff);
    END_IF;

    IF wait720.top AND NOT (pnsWaitOff.top) THEN
          testUnsuccessfulUnfill.error:=TRUE;
    END_IF;

    IF pnsWaitOff.top THEN
          resetPhase(wait720);
	waitReset(IN:=TRUE, PT:= T#3S);
    END_IF;

    IF waitReset.Q THEN
        resetIfRunning(algoritms.vibegPNS);
        algManager.nMode:=ModeGpa.MODE_STOP;
        resetIfRunning(StrAlg);
    END_IF;

    StrAlg.isEnded:= pnsWaitOff.top;

    IF OpcCommandsKransEnabled AND NOT OpcCommandsKransDisabled THEN
	IF      (im.pns.onStatus = _statusDualInput.STATUS_ON)
              AND (im.nu1.onStatus = _statusDualInput.STATUS_ON OR im.nu2.onStatus = _statusDualInput.STATUS_ON)
	    AND (ai.Tmasla_MB.interval >= _statusAi.normal)
              (*AND (ai.Tmasla_MB.value > im.PuskOilSystem_UstdPmg.Value)*)
          THEN
	    IM.Kran3b.inOpcCommandsDisabled:=FALSE;
	    Im.kran4.inOpcCommandsDisabled:=FALSE;
	    Im.kran5.inOpcCommandsDisabled:=FALSE;
		(*IF	Im.SingleSignals.dP_gazgaz_Kran1.q THEN
			Im.kran1.inOpcCommandsDisabled:=FALSE;
			Im.kran2.inOpcCommandsDisabled:=FALSE;
		ELSE
			Im.kran1.inOpcCommandsDisabled:=TRUE;
			Im.kran2.inOpcCommandsDisabled:=TRUE;
		END_IF;*)
          ELSE
	    Im.kran1.inOpcCommandsDisabled:=TRUE;
	    Im.kran2.inOpcCommandsDisabled:=TRUE;
	    Im.kran3b.inOpcCommandsDisabled:=TRUE;
	    Im.kran4.inOpcCommandsDisabled:=TRUE;
	    Im.kran5.inOpcCommandsDisabled:=TRUE;
          END_IF;

    ELSE
	Im.kran1.inOpcCommandsDisabled:=TRUE;
	Im.kran2.inOpcCommandsDisabled:=TRUE;
	Im.kran3b.inOpcCommandsDisabled:=TRUE;
	Im.kran4.inOpcCommandsDisabled:=TRUE;
	Im.kran5.inOpcCommandsDisabled:=TRUE;
    END_IF;
END_IF;

StrAlg.CanRun := StrAlg.inCanRun;
StrAlg.OpcCommandsDisabled := StrAlg.inOpcCommandsDisabled;

(* ---- Если управление с ВУ заблокировано, то  передаем команду из алгоритма ---- *)
IF StrAlg.inOpcCommandsDisabled THEN
	StrAlg.inCommand := StrAlg.inCommand_Alg;
ELSE (* иначе передаем команду с АРМа*)
	StrAlg.inCommand := StrAlg.inCommand_ARM;
END_IF;

_sunpackerCommand(command := StrAlg.inCommand);
	source := _sunpackerCommand.source;
	cmd := _sunpackerCommand.cmd;

IF cmd <> 0 AND lastCmd <> cmd AND (((NOT StrAlg.opcCommandsDisabled) AND source > 0) OR source = 0) then
	CASE BYTE_TO_INT(cmd) OF
		(*cmdRun*) 1: 	IF (StrAlg.CanRun) THEN
					StrAlg.isRuning := TRUE;
					StrAlg.isEnded := FALSE;
					StrAlg.hasError := FALSE;
					(*****************       OnRun       *****************)

                                                  algManager.nMode:=ModeGpa.MODE_PUSKK;
                                                  resetAndDisable(alg:=algoritms.ppu);
                                                  algoritms.puskOilSystem.inCanRun:= TRUE;
                                                  algoritms.filling.inCanRun:= TRUE;
                                                  runPhase(puskOilSystem);

					cmd_for_Status := cmd;
					source_for_Status := source;
					command_error_for_Status := 0;
				ELSE
					StrAlg.isRuning := FALSE;
					StrAlg.isEnded := FALSE;
					StrAlg.hasError 	:= FALSE;

					cmd_for_Status := 0;
					source_for_Status := source;
					command_error_for_Status := cmd;
				END_IF;
		(*cmdReset*) 2: 	StrAlg.isRuning := FALSE;
				StrAlg.isEnded := FALSE;
				StrAlg.hasError 	:= FALSE;

                                         (*****************       OnReset       *****************)
                                        OpcCommandsKransEnabled:=FALSE;
                                        OpcCommandsKransDisabled:=FALSE;
                                        waitReset(IN:=FALSE);
                                        _resetQuestion1:=FALSE;
                                        _resetQuestion2:=FALSE;
                                        resetPhase(puskOilSystem);
                                        resetPhase(filling);
                                        resetPhase(kran3bOpen);
                                        resetPhase(kran4Close);
                                        resetPhase(kran1Close);
                                        resetPhase(kran2Close);
                                        resetPhase(kran5open);
                                        resetPhase(wait720);
                                        resetPhase(noGasInPipe);
                                        resetPhase(AutoNUoff);
                                        resetPhase(nu1Off);
                                        resetPhase(nu2Off);
                                        resetPhase(pnsWaitOff);
                                        resetPhase(testUnsuccessfulUnfill);
                                        BlockAllIM(IM);
                                        resetQuestion(questionFilling);
                                        resetQuestion(questionUnload);

                                        StrAlg.inOpcCommandsDisabled:=FALSE;

				cmd_for_Status := cmd;
				source_for_Status := source;
				command_error_for_Status := 0;
	END_CASE;
	resetCmdTimer(IN := false);
	resetCmdTimerPriznak := TRUE;
END_IF;
lastCmd := cmd;

resetCmdTimer(IN := resetCmdTimerPriznak, PT := T#5S);
IF resetCmdTimer.Q THEN
	resetCmdTimerPriznak := FALSE;
	source_for_Status := 0;
	cmd_for_Status := 0;
	command_error_for_Status := 0;
END_IF;

StrAlg.Start:= puskOilSystem.startStatus
            OR filling.startStatus
            OR kran3bOpen.startStatus
            OR kran4Close.startStatus
            OR kran1Close.startStatus
            OR kran2Close.startStatus
            OR kran5open.startStatus
            OR wait720.startStatus
            OR noGasInPipe.startStatus
            OR AutoNUoff.startStatus
            OR nu1Off.startStatus
            OR nu2Off.startStatus
            OR pnsWaitOff.startStatus
            OR testUnsuccessfulUnfill.startStatus;

StrAlg.Error:=  puskOilSystem.errorStatus
            OR filling.errorStatus
            OR kran3bOpen.errorStatus
            OR kran4Close.errorStatus
            OR kran1Close.errorStatus
            OR kran2Close.errorStatus
            OR kran5open.errorStatus
            OR wait720.errorStatus
            OR noGasInPipe.errorStatus
            OR AutoNUoff.errorStatus
            OR nu1Off.errorStatus
            OR nu2Off.errorStatus
            OR pnsWaitOff.errorStatus
            OR testUnsuccessfulUnfill.errorStatus;

StrAlg.Top:=   puskOilSystem.topStatus
            OR filling.topStatus
            OR kran3bOpen.topStatus
            OR kran4Close.topStatus
            OR kran1Close.topStatus
            OR kran2Close.topStatus
            OR kran5open.topStatus
            OR wait720.topStatus
            OR noGasInPipe.topStatus
            OR AutoNUoff.topStatus
            OR nu1Off.topStatus
            OR nu2Off.topStatus
            OR pnsWaitOff.topStatus
            OR testUnsuccessfulUnfill.topStatus;

(*TODO: TYPE PROGRAM CODE HERE*)
StrAlg.status :=  SHL(BYTE_TO_DWORD(source_for_Status), 29)
			OR SHL(BYTE_TO_DWORD(cmd_for_Status), 26)
			OR SHL(BYTE_TO_DWORD(command_error_for_Status), 23)
			OR SHL(BOOL_TO_DWORD(StrAlg.OpcCommandsDisabled ), 21)
			OR SHL(BOOL_TO_DWORD(StrAlg.hasError),4)
			OR SHL(BOOL_TO_DWORD(StrAlg.CanRun),2)
			OR SHL(BOOL_TO_DWORD(StrAlg.isEnded),1)
			OR BOOL_TO_DWORD(StrAlg.isRuning);

(* ---- puskValg.st ---- *)
FUNCTION_BLOCK puskValg

VAR_IN_OUT
	StrAlg : struct_Alg;
END_VAR

VAR
	puskOilSystem : struct_PhaseAlgoritm;
END_VAR

VAR_IN_OUT
	questionEngine : struct_Question;
END_VAR

VAR
	runningEngine : struct_PhaseAlgoritm;
END_VAR

VAR_IN_OUT
	questionMVoff : struct_Question;
END_VAR

VAR
	mvOff : struct_PhaseAlgoritm;
	pnsOn : struct_PhaseAlgoritm;
	wait600 : struct_PhaseAlgoritm;
	AutoNUoff : struct_PhaseAlgoritm;
	nu1Off : struct_PhaseAlgoritm;
	nu2Off : struct_PhaseAlgoritm;
	autoAvomOff : struct_PhaseAlgoritm;
	Avom1Off : struct_PhaseAlgoritm;
	Avom2Off : struct_PhaseAlgoritm;
	pnsWaitOff : struct_PhaseAlgoritm;
	testUnsuccessful : struct_PhaseAlgoritm;
	fb_puskOilSystem : fb_ph_algoritm;
	fb_questionEngine : fb_Question;
	fb_runningEngine : fb_ph_algoritm;
	fb_questionMVoff : fb_Question;
	fb_mvOff : fb_ph_SectionSwitch;
	fb_pnsOn : fb_ph_Switch;
	fb_wait600 : fb_ph_Timer;
	fb_AutoNUoff : fb_ph_algoritm;
	fb_nu1Off : fb_ph_OilPump;
	fb_nu2Off : fb_ph_OilPump;
	fb_autoAvomOff : fb_ph_algoritm;
	fb_Avom1Off : fb_ph_Switch;
	fb_Avom2Off : fb_ph_Switch;
	fb_pnsWaitOff : fb_ph_algoritm;
	fb_testUnsuccessful : fb_ph_CustomPhase;
	_sunpackerCommand : fb_sunpackerCommand;
	_DualStateImAction : TYPE_DualStateImAction;
	_Answers : TYPE_Answers;
	_statusDualInput : TYPE_statusDualInput;
	_StatusAi : TYPE_StatusAi;
	_PhaseAlgoritmAction : TYPE_PhaseAlgoritmAction;
	source : BYTE;
	cmd : BYTE;
	lastCmd : BYTE;
	source_for_Status : BYTE;
	cmd_for_Status : BYTE;
	command_error_for_Status : BYTE;
	resetCmdTimer : TON;
	resetCmdTimerPriznak : BOOL;
	onInit : BOOL;
	_resetQuestion1 : BOOL;
	_resetQuestion2 : BOOL;
	waitReset : TON;
END_VAR

VAR_EXTERNAL
	IM : ImConfig;
	algoritms : AlgoritmsConfig;
	ai : AiConfig;
	AlgTimers : struct_AlgTimers;
	ModeGpa : TYPE_ModeGpa;
	algManager : struct_AlgoritmsManager;
	protections : ProtectionsConfig;
END_VAR

VAR CONSTANT
	Ust_Pgaza : LREAL          := 0.3;
END_VAR

IF NOT onInit THEN

          fb_puskOilSystem(phaseNumber:=0, act:=_run, waitCompletion:=TRUE);
       questionEngine.AnswerVariants:=_Answers.ANS_YES;
          fb_runningEngine(phaseNumber:=1, act:=_run, waitCompletion:=TRUE);
        questionMVoff.AnswerVariants:=_Answers.ANS_YES;
                  fb_mvOff(phaseNumber:=3, act:=_off);
                  fb_pnsOn(phaseNumber:=4, act:=_on);
                fb_wait600(phaseNumber:=8, delay:=T#600S);
              fb_AutoNUoff(phaseNumber:=10, act:=_reset, waitCompletion:=FALSE);
                 fb_nu1Off(phaseNumber:=11, act:=_off);
                 fb_nu2Off(phaseNumber:=12, act:=_off);
             fb_pnsWaitOff(phaseNumber:=15, act:=_run, waitCompletion:=TRUE);
            fb_autoAvomOff(phaseNumber:=7, act:=_reset, waitCompletion:=FALSE);
               fb_Avom1Off(phaseNumber:=5, act:=_off);
               fb_Avom2Off(phaseNumber:=6, act:=_off);
       fb_testUnsuccessful(phaseNumber:=17);

onInit:=TRUE;
END_IF;

          fb_puskOilSystem(StrPh:=puskOilSystem, alg:=algoritms.puskOilSystem);
         fb_questionEngine(StrQ:=questionEngine);
          fb_runningEngine(StrPh:=runningEngine, alg:=algoritms.engineRun);
          fb_questionMVoff(StrQ:=questionMVoff);
                  fb_mvOff(StrPh:=mvOff, Im:=Im.mv);
                  fb_pnsOn(StrPh:=pnsOn, Im:=Im.pns);
                fb_wait600(StrPh:=wait600, timer:=AlgTimers.puskV_wait600);
              fb_AutoNUoff(StrPh:=AutoNUoff, alg:=algoritms.autoNu);
                 fb_nu1Off(StrPh:=nu1Off, Im:=Im.nu1);
                 fb_nu2Off(StrPh:=nu2Off, Im:=Im.nu2);
             fb_pnsWaitOff(StrPh:=pnsWaitOff, alg:=algoritms.vibegPNS);
            fb_autoAvomOff(StrPh:=autoAvomOff, alg:=algoritms.AutoAvom);
               fb_Avom1Off(StrPh:=Avom1Off, Im:=Im.v1_Avom);
               fb_Avom2Off(StrPh:=Avom2Off, Im:=Im.v2_Avom);
       fb_testUnsuccessful(StrPh:=testUnsuccessful);

StrAlg.CanRun := StrAlg.inCanRun;
StrAlg.OpcCommandsDisabled := StrAlg.inOpcCommandsDisabled;

IF StrAlg.isRuning THEN

    StrAlg.hasError := mvOff.error OR pnsOn.error OR testUnsuccessful.error;

    IF puskOilSystem.top THEN
         IF NOT _resetQuestion1 THEN
         askQuestion(questionEngine);
         _resetQuestion1:=TRUE;
         END_IF;
    END_IF;

    IF questionEngine.answer = _Answers.ANS_YES THEN
        runPhase(runningEngine);
        resetQuestion(questionEngine);
    END_IF;

    IF runningEngine.top THEN
       IF NOT _resetQuestion2 THEN
       askQuestion(questionMVoff);
       _resetQuestion2:=TRUE;
       END_IF;
    END_IF;

     IF questionMVoff.answer = _Answers.ANS_YES THEN

        (*resetDiProtection(protections.Pgaza_na_vyhode_nagnetatelia_GPA_STOP);
       *) resetIfRunning(algoritms.AutoPns);
        runPhase(mvOff);
        runPhase(wait600);
        resetQuestion(questionMVoff);
     END_IF;

    IF mvOff.top THEN
        runPhase(pnsOn);
    END_IF;

    IF pnsOn.top THEN

          ai.Tmasla_MB.Disabled_LA:=TRUE;
          ai.Tmasla_MB.Disabled_LW:=TRUE;
          (*IM.SingleSignals.dP_oilgaz_low.Disabled_Sig:=TRUE;*)
          (*resetAiProtection(protections.Os_sdvig_nagnetatelja_plus)*)
         (* resetDiProtection(protections.Vibro_skorost_OP_shesterni_RED_T5);*)
	runPhase(AutoNUoff);

    END_IF;

     IF autoNuOff.top THEN
	runPhase(nu1off);
          runPhase(nu2off);
    END_IF;

    IF nu1Off.top AND nu2Off.top THEN
	runPhase(pnsWaitOff);
    END_IF;

    IF wait600.top AND NOT (pnsWaitOff.top) THEN
          testUnsuccessful.error:=TRUE;
    END_IF;

    IF pnsWaitOff.top THEN
          resetPhase(wait600);
          runPhase(autoAvomOff);
	waitReset(IN:=TRUE, PT:= T#3S);
    END_IF;

    IF autoAvomOff.top THEN
          runPhase(Avom1Off);
          runPhase(Avom2Off);
    END_IF;

    IF waitReset.Q THEN
        resetIfRunning(algoritms.vibegPNS);
        algManager.nMode:=ModeGpa.MODE_STOP;
        resetIfRunning(StrAlg);
    END_IF;

    StrAlg.isEnded:= pnsWaitOff.top;

END_IF;

StrAlg.CanRun := StrAlg.inCanRun;
StrAlg.OpcCommandsDisabled := StrAlg.inOpcCommandsDisabled;

(* ---- Если управление с ВУ заблокировано, то  передаем команду из алгоритма ---- *)
IF StrAlg.inOpcCommandsDisabled THEN
	StrAlg.inCommand := StrAlg.inCommand_Alg;
ELSE (* иначе передаем команду с АРМа*)
	StrAlg.inCommand := StrAlg.inCommand_ARM;
END_IF;

_sunpackerCommand(command := StrAlg.inCommand);
	source := _sunpackerCommand.source;
	cmd := _sunpackerCommand.cmd;

IF cmd <> 0 AND lastCmd <> cmd AND (((NOT StrAlg.opcCommandsDisabled) AND source > 0) OR source = 0) then
	CASE BYTE_TO_INT(cmd) OF
		(*cmdRun*) 1: 	IF (StrAlg.CanRun) THEN
					StrAlg.isRuning := TRUE;
					StrAlg.isEnded := FALSE;
					StrAlg.hasError := FALSE;
					(*****************       OnRun       *****************)

                                                  algManager.nMode:=ModeGpa.MODE_PUSKV;
                                                  resetAndDisable(alg:=algoritms.ppu);
                                                  algoritms.puskOilSystem.inCanRun:= TRUE;
                                                  algoritms.engineRun.inCanRun:= TRUE;
                                                  runPhase(puskOilSystem);

					cmd_for_Status := cmd;
					source_for_Status := source;
					command_error_for_Status := 0;
				ELSE
					StrAlg.isRuning := FALSE;
					StrAlg.isEnded := FALSE;
					StrAlg.hasError 	:= FALSE;

					cmd_for_Status := 0;
					source_for_Status := source;
					command_error_for_Status := cmd;
				END_IF;
		(*cmdReset*) 2: 	StrAlg.isRuning := FALSE;
				StrAlg.isEnded := FALSE;
				StrAlg.hasError 	:= FALSE;

                                         (*****************       OnReset       *****************)
                                        waitReset(IN:=FALSE);
                                        _resetQuestion1:=FALSE;
                                        _resetQuestion2:=FALSE;
                                        resetPhase(puskOilSystem);
                                        resetPhase(runningEngine);
                                        resetPhase(mvOff);
                                        resetPhase(pnsOn);
                                        resetPhase(wait600);
                                        resetPhase(AutoNUoff);
                                        resetPhase(nu1Off);
                                        resetPhase(nu2Off);
                                        resetPhase(pnsWaitOff);
	                              resetPhase(autoAvomOff);
                                        resetPhase(Avom1Off);
                                        resetPhase(Avom2Off);
                                        resetPhase(testUnsuccessful);

                                        resetQuestion(questionEngine);
                                        resetQuestion(questionMVoff);

                                        StrAlg.inOpcCommandsDisabled:=FALSE;

				cmd_for_Status := cmd;
				source_for_Status := source;
				command_error_for_Status := 0;
	END_CASE;
	resetCmdTimer(IN := false);
	resetCmdTimerPriznak := TRUE;
END_IF;
lastCmd := cmd;

resetCmdTimer(IN := resetCmdTimerPriznak, PT := T#5S);
IF resetCmdTimer.Q THEN
	resetCmdTimerPriznak := FALSE;
	source_for_Status := 0;
	cmd_for_Status := 0;
	command_error_for_Status := 0;
END_IF;

StrAlg.Start:= puskOilSystem.startStatus
            OR runningEngine.startStatus
            OR mvOff.startStatus
            OR pnsOn.startStatus
            OR wait600.startStatus
            OR AutoNUoff.startStatus
            OR nu1Off.startStatus
            OR nu2Off.startStatus
            OR pnsWaitOff.startStatus
            OR testUnsuccessful.startStatus;

StrAlg.Error:=  puskOilSystem.errorStatus
            OR runningEngine.errorStatus
            OR mvOff.errorStatus
            OR pnsOn.errorStatus
            OR wait600.errorStatus
            OR AutoNUoff.errorStatus
            OR nu1Off.errorStatus
            OR nu2Off.errorStatus
            OR pnsWaitOff.errorStatus
            OR testUnsuccessful.errorStatus;

StrAlg.Top:=   puskOilSystem.topStatus
            OR runningEngine.topStatus
            OR mvOff.topStatus
            OR pnsOn.topStatus
            OR wait600.topStatus
            OR AutoNUoff.topStatus
            OR nu1Off.topStatus
            OR nu2Off.topStatus
            OR pnsWaitOff.topStatus
            OR testUnsuccessful.topStatus;

(*TODO: TYPE PROGRAM CODE HERE*)
StrAlg.status :=  SHL(BYTE_TO_DWORD(source_for_Status), 29)
			OR SHL(BYTE_TO_DWORD(cmd_for_Status), 26)
			OR SHL(BYTE_TO_DWORD(command_error_for_Status), 23)
			OR SHL(BOOL_TO_DWORD(StrAlg.OpcCommandsDisabled ), 21)
			OR SHL(BOOL_TO_DWORD(StrAlg.hasError),4)
			OR SHL(BOOL_TO_DWORD(StrAlg.CanRun),2)
			OR SHL(BOOL_TO_DWORD(StrAlg.isEnded),1)
			OR BOOL_TO_DWORD(StrAlg.isRuning);

(* ---- RemontAlg.st ---- *)
FUNCTION_BLOCK RemontAlg

VAR_IN_OUT
	StrAlg : struct_Alg;
END_VAR

VAR
	_sunpackerCommand : fb_sunpackerCommand;
	source : BYTE;
	cmd : BYTE;
	lastCmd : BYTE;
	source_for_Status : BYTE;
	cmd_for_Status : BYTE;
	command_error_for_Status : BYTE;
	resetCmdTimer : TON;
	resetCmdTimerPriznak : BOOL;
END_VAR

VAR_EXTERNAL
	protectManager : struct_ProtectionsManager;
	algManager : struct_AlgoritmsManager;
	ModeGpa : TYPE_ModeGpa;
	PMcommand : TYPE_CommandsPotectionsManager;
	IM : ImConfig;
END_VAR

StrAlg.CanRun := StrAlg.inCanRun;
StrAlg.OpcCommandsDisabled := StrAlg.inOpcCommandsDisabled;

(* ---- Если управление с ВУ заблокировано, то передаем команду из алгоритма ---- *)
IF StrAlg.inOpcCommandsDisabled THEN
	StrAlg.inCommand := StrAlg.inCommand_Alg;
ELSE (* иначе передаем команду с АРМа*)
	StrAlg.inCommand := StrAlg.inCommand_ARM;
END_IF;

_sunpackerCommand(command := StrAlg.inCommand);
	source := _sunpackerCommand.source;
	cmd := _sunpackerCommand.cmd;

IF cmd <> 0 AND lastCmd <> cmd AND (((NOT StrAlg.opcCommandsDisabled) AND source > 0) OR source = 0) then
	CASE BYTE_TO_INT(cmd) OF
		(*cmdRun*) 1: 	IF (StrAlg.CanRun) THEN
					StrAlg.isRuning := TRUE;
					StrAlg.isEnded := FALSE;
					StrAlg.hasError 	:= FALSE;
                                             (*****************       OnRun       *****************)
                                                      algManager.nMode:=ModeGpa.MODE_REMONT;
                                                      protectManager.inCommand:=PMcommand.ResetAllProtections;
					    UnBlockAllIM(IM);
                                                  (*StrAlg.inOpcCommandsDisabled:=FALSE;*)
					cmd_for_Status := cmd;
					source_for_Status := source;
					command_error_for_Status := 0;
				ELSE
					StrAlg.isRuning := FALSE;
					StrAlg.isEnded := FALSE;
					StrAlg.hasError 	:= FALSE;

					cmd_for_Status := 0;
					source_for_Status := source;
					command_error_for_Status := cmd;
				END_IF;
		(*cmdReset*) 2: 	StrAlg.isRuning := FALSE;
				StrAlg.isEnded := FALSE;
				StrAlg.hasError 	:= FALSE;
                                        (*****************       OnReset       *****************)
                                                  BlockAllIM(IM);
                                                  protectManager.inCommand:=PMcommand.RestartAllProtections;
                                                  algManager.nMode:=ModeGpa.MODE_STOP;

				cmd_for_Status := cmd;
				source_for_Status := source;
				command_error_for_Status := 0;
	END_CASE;
	resetCmdTimer(IN := false);
	resetCmdTimerPriznak := TRUE;
END_IF;
lastCmd := cmd;

resetCmdTimer(IN := resetCmdTimerPriznak, PT := T#5S);
IF resetCmdTimer.Q THEN
	resetCmdTimerPriznak := FALSE;
	source_for_Status := 0;
	cmd_for_Status := 0;
	command_error_for_Status := 0;
END_IF;

StrAlg.status :=  SHL(BYTE_TO_DWORD(source_for_Status), 29)
			OR SHL(BYTE_TO_DWORD(cmd_for_Status), 26)
			OR SHL(BYTE_TO_DWORD(command_error_for_Status), 23)
			OR SHL(BOOL_TO_DWORD(StrAlg.OpcCommandsDisabled ), 21)
			OR SHL(BOOL_TO_DWORD(StrAlg.hasError),4)
			OR SHL(BOOL_TO_DWORD(StrAlg.CanRun),2)
			OR SHL(BOOL_TO_DWORD(StrAlg.isEnded),1)
			OR BOOL_TO_DWORD(StrAlg.isRuning);

(* ---- SemiAutoPuskAlg.st ---- *)
FUNCTION_BLOCK SemiAutoPuskAlg

VAR_IN_OUT
	StrAlg : struct_Alg;
END_VAR

VAR
	runOilsystem : struct_PhaseAlgoritm;
	runEngine : struct_PhaseAlgoritm;
	filling : struct_PhaseAlgoritm;
END_VAR

VAR_IN_OUT
	cmdRun1ph : struct_Question;
	cmdRun2ph : struct_Question;
	cmdRun3ph : struct_Question;
END_VAR

VAR
	fb_runOilsystem : fb_ph_algoritm;
	fb_runEngine : fb_ph_algoritm;
	fb_filling : fb_ph_algoritm;
	fb_cmdRun1ph : fb_Question;
	fb_cmdRun2ph : fb_Question;
	fb_cmdRun3ph : fb_Question;
	_sunpackerCommand : fb_sunpackerCommand;
	_PhaseAlgoritmAction : TYPE_PhaseAlgoritmAction;
	_statusDualInput : TYPE_statusDualInput;
	_Answers : TYPE_Answers;
	source : BYTE;
	cmd : BYTE;
	lastCmd : BYTE;
	source_for_Status : BYTE;
	cmd_for_Status : BYTE;
	command_error_for_Status : BYTE;
	resetCmdTimer : TON;
	resetCmdTimerPriznak : BOOL;
	onInit : BOOL;
	waitReset : TON;
END_VAR

VAR_EXTERNAL
	algoritms : AlgoritmsConfig;
	ModeGpa : TYPE_ModeGpa;
	algManager : struct_AlgoritmsManager;
	IM : ImConfig;
END_VAR

IF NOT onInit THEN
               cmdRun1ph.AnswerVariants:=_Answers.ANS_YES;
         fb_runOilsystem(phaseNumber:=0, act:=_run, waitCompletion:=TRUE);
               cmdRun2ph.AnswerVariants:=_Answers.ANS_YES;
            fb_runEngine(phaseNumber:=1, act:=_run, waitCompletion:=TRUE);
               cmdRun3ph.AnswerVariants:=_Answers.ANS_YES;
              fb_filling(phaseNumber:=2, act:=_run, waitCompletion:=TRUE);

onInit:=TRUE;
END_IF;
            fb_cmdRun1ph(StrQ:=cmdRun1ph);
         fb_runOilsystem(StrPh:=runOilsystem, alg:=algoritms.puskOilSystem);
            fb_cmdRun2ph(StrQ:=cmdRun2ph);
            fb_runEngine(StrPh:=runEngine, alg:=algoritms.engineRun);
            fb_cmdRun3ph(StrQ:=cmdRun3ph);
              fb_filling(StrPh:=filling, alg:=algoritms.filling);

StrAlg.CanRun := StrAlg.inCanRun;
StrAlg.OpcCommandsDisabled := StrAlg.inOpcCommandsDisabled;

IF StrAlg.isRuning THEN

    StrAlg.hasError := runOilsystem.error OR runEngine.error OR filling.error;

    IF cmdRun1ph.answer = _Answers.ANS_YES THEN
	runPhase(runOilsystem);
          resetQuestion(cmdRun1ph);
    END_IF;

    IF runOilsystem.top AND NOT runEngine.start THEN
         askQuestion(cmdRun2ph);
    END_IF;

    IF cmdRun2ph.answer = _Answers.ANS_YES THEN
         runPhase(runEngine);
         resetQuestion(cmdRun2ph);
    END_IF;

    IF runEngine.top AND NOT filling.start THEN
         askQuestion(cmdRun3ph);
    END_IF;

    IF cmdRun3ph.answer = _Answers.ANS_YES THEN
         runPhase(filling);
         resetQuestion(cmdRun3ph);
    END_IF;

    IF filling.top THEN
          waitReset(IN:=TRUE, PT:= T#2S);
    END_IF;

    IF waitReset.Q THEN

        IF Im.kran6.onStatus = _statusDualInput.STATUS_On THEN
	algManager.nMode:= ModeGpa.MODE_WORK_Ring;
        END_IF;
        IF Im.kran6.onStatus = _statusDualInput.STATUS_Off THEN
	algManager.nMode:= ModeGpa.MODE_WORK_Line;
        END_IF;

        resetIfRunning(StrAlg);
    END_IF;

    StrAlg.isEnded:= filling.top;

END_IF;

StrAlg.CanRun := StrAlg.inCanRun;
StrAlg.OpcCommandsDisabled := StrAlg.inOpcCommandsDisabled;

(* ---- Если управление с ВУ заблокировано, то  передаем команду из алгоритма ---- *)
IF StrAlg.inOpcCommandsDisabled THEN
	StrAlg.inCommand := StrAlg.inCommand_Alg;
ELSE (* иначе передаем команду с АРМа*)
	StrAlg.inCommand := StrAlg.inCommand_ARM;
END_IF;

_sunpackerCommand(command := StrAlg.inCommand);
	source := _sunpackerCommand.source;
	cmd := _sunpackerCommand.cmd;

IF cmd <> 0 AND lastCmd <> cmd AND (((NOT StrAlg.opcCommandsDisabled) AND source > 0) OR source = 0) then
	CASE BYTE_TO_INT(cmd) OF
		(*cmdRun*) 1: 	IF (StrAlg.CanRun) THEN
					StrAlg.isRuning := TRUE;
					StrAlg.isEnded := FALSE;
					StrAlg.hasError := FALSE;
					(*****************       OnRun       *****************)

                                                  algoritms.puskOilSystem.inCanRun:= TRUE	;
                                                  algoritms.filling.inCanRun:= TRUE	;
                                                  algoritms.engineRun.inCanRun:= TRUE	;

                                                  algManager.nMode:=ModeGpa.MODE_MPUSK;
                                                  (*impulseSO(Im.SingleOutputs.VzvodBREO);*)
                                                  askQuestion(cmdRun1ph);

					cmd_for_Status := cmd;
					source_for_Status := source;
					command_error_for_Status := 0;
				ELSE
					StrAlg.isRuning := FALSE;
					StrAlg.isEnded := FALSE;
					StrAlg.hasError 	:= FALSE;

					cmd_for_Status := 0;
					source_for_Status := source;
					command_error_for_Status := cmd;
				END_IF;
		(*cmdReset*) 2: 	StrAlg.isRuning := FALSE;
				StrAlg.isEnded := FALSE;
				StrAlg.hasError 	:= FALSE;

                                         (*****************       OnReset       *****************)
                                        waitReset(IN:=FALSE);
                                        StrAlg.inCanRun:=FALSE;

                                        resetPhase(runOilsystem);
                                        resetPhase(runEngine);
                                        resetPhase(filling);

                                        resetQuestion(cmdRun1ph);
                                        resetQuestion(cmdRun2ph);
                                        resetQuestion(cmdRun3ph);

                                        StrAlg.inOpcCommandsDisabled:=FALSE;

				cmd_for_Status := cmd;
				source_for_Status := source;
				command_error_for_Status := 0;
	END_CASE;
	resetCmdTimer(IN := false);
	resetCmdTimerPriznak := TRUE;
END_IF;
lastCmd := cmd;

resetCmdTimer(IN := resetCmdTimerPriznak, PT := T#5S);
IF resetCmdTimer.Q THEN
	resetCmdTimerPriznak := FALSE;
	source_for_Status := 0;
	cmd_for_Status := 0;
	command_error_for_Status := 0;
END_IF;

StrAlg.Start:= runOilsystem.startStatus
            OR runEngine.startStatus
            OR filling.startStatus;

StrAlg.Error:= runOilsystem.errorStatus
            OR runEngine.errorStatus
            OR filling.errorStatus;

StrAlg.Top:=   runOilsystem.topStatus
            OR runEngine.topStatus
            OR filling.topStatus;

(*TODO: TYPE PROGRAM CODE HERE*)
StrAlg.status :=  SHL(BYTE_TO_DWORD(source_for_Status), 29)
			OR SHL(BYTE_TO_DWORD(cmd_for_Status), 26)
			OR SHL(BYTE_TO_DWORD(command_error_for_Status), 23)
			OR SHL(BOOL_TO_DWORD(StrAlg.OpcCommandsDisabled ), 21)
			OR SHL(BOOL_TO_DWORD(StrAlg.hasError),4)
			OR SHL(BOOL_TO_DWORD(StrAlg.CanRun),2)
			OR SHL(BOOL_TO_DWORD(StrAlg.isEnded),1)
			OR BOOL_TO_DWORD(StrAlg.isRuning);

(* ---- testdPmgAlg.st ---- *)
FUNCTION_BLOCK testdPmgAlg

VAR_IN_OUT
	StrAlg : struct_Alg;
END_VAR

VAR
	puskOilSystem : struct_PhaseAlgoritm;
END_VAR

VAR_IN_OUT
	algContinue : struct_Question;
END_VAR

VAR
	nuOff : struct_PhaseAlgoritm;
	dPmgAi : struct_PhaseAlgoritm;
	dPmgDi : struct_PhaseAlgoritm;
	nuOn : struct_PhaseAlgoritm;
	noRezrv : struct_PhaseAlgoritm;
	BreakTest : struct_PhaseAlgoritm;
	testUnsuccessful : struct_PhaseAlgoritm;
	pnsOff : struct_PhaseAlgoritm;
	stopANU : struct_PhaseAlgoritm;
	Ust_dPLow : struct_PhaseAlgoritm;
	nu1Off : struct_PhaseAlgoritm;
	nu2Off : struct_PhaseAlgoritm;
	stopNU1 : struct_PhaseAlgoritm;
	stopNU2 : struct_PhaseAlgoritm;
	fb_puskOilSystem : fb_ph_algoritm;
	fb_algContinue : fb_Question;
	fb_nuOff : fb_ph_CustomPhase;
	fb_dPmgAi : fb_ph_WaitAnalogValue;
	fb_dPmgDi : fb_ph_CustomPhase;
	fb_nuOn : fb_ph_CustomPhase;
	fb_noRezrv : fb_ph_CustomPhase;
	fb_BreakTest : fb_ph_Timer;
	fb_testUnsuccessful : fb_ph_CustomPhase;
	fb_pnsOff : fb_ph_Switch;
	fb_stopANU : fb_ph_CustomPhase;
	fb_nu1Off : fb_ph_OilPump;
	fb_nu2Off : fb_ph_OilPump;
	fb_stopNU1 : fb_ph_OilPump;
	fb_stopNU2 : fb_ph_OilPump;
	_sunpackerCommand : fb_sunpackerCommand;
	_DualStateImAction : TYPE_DualStateImAction;
	_Answers : TYPE_Answers;
	_statusDualInput : TYPE_statusDualInput;
	_StatusAi : TYPE_StatusAi;
	_PhaseAlgoritmAction : TYPE_PhaseAlgoritmAction;
	source : BYTE;
	cmd : BYTE;
	lastCmd : BYTE;
	source_for_Status : BYTE;
	cmd_for_Status : BYTE;
	command_error_for_Status : BYTE;
	resetCmdTimer : TON;
	resetCmdTimerPriznak : BOOL;
	onInit : BOOL;
	_resetQuestion : BOOL;
	waitReset : TON;
	WaitOnNU : TON;
END_VAR

VAR_EXTERNAL
	IM : ImConfig;
	algoritms : AlgoritmsConfig;
	ai : AiConfig;
	AlgTimers : struct_AlgTimers;
	ModeGpa : TYPE_ModeGpa;
	algManager : struct_AlgoritmsManager;
	protections : ProtectionsConfig;
	NotHasRezervNU : BOOL;
END_VAR

IF NOT onInit THEN

    fb_puskOilSystem(phaseNumber:=0, act:=_run, waitCompletion:=TRUE);
        algContinue.AnswerVariants:=_Answers.ANS_YES;
            fb_nuOff(phaseNumber:=1);
           fb_dPmgAi(phaseNumber:=2);
           fb_dPmgDi(phaseNumber:=3);
             fb_nuOn(phaseNumber:=4);
          fb_noRezrv(phaseNumber:=5);
 fb_testUnsuccessful(phaseNumber:=6);
        fb_BreakTest(phaseNumber:=7, delay:=T#10S);
           fb_pnsOff(phaseNumber:=8, act:=_off);
          fb_stopANU(phaseNumber:=9);
           fb_nu1Off(phaseNumber:=11, act:=_off);
           fb_nu2Off(phaseNumber:=12, act:=_off);
          fb_stopNU1(phaseNumber:=15, act:=_off);
          fb_stopNU2(phaseNumber:=16, act:=_off);
onInit:=TRUE;
END_IF;

    fb_puskOilSystem(StrPh:=puskOilSystem, alg:=algoritms.puskOilSystem);
      fb_algContinue(StrQ:=algContinue);
            fb_nuOff(StrPh:=nuOff);
           (*fb_dPmgAi(StrPh:=dPmgAi, ai:=ai.Tmasla_MB, less:=im.testdPmg_Ust_dPLow.Value);*)
           fb_dPmgDi(StrPh:=dPmgDi);
             fb_nuOn(StrPh:=nuOn);
          fb_noRezrv(StrPh:=noRezrv);
 fb_testUnsuccessful(StrPh:=testUnsuccessful);
        fb_BreakTest(StrPh:=BreakTest, timer:=AlgTimers.testdPmg_BreakTest);
           fb_pnsOff(StrPh:=pnsOff, Im:=Im.pns);
          fb_stopANU(StrPh:=stopANU);
           fb_nu1Off(StrPh:=nu1Off, Im:=Im.nu1);
           fb_nu2Off(StrPh:=nu2Off, Im:=Im.nu2);
          fb_stopNU1(StrPh:=stopNU1, Im:=Im.nu1);
          fb_stopNU2(StrPh:=stopNU2, Im:=Im.nu2);

StrAlg.CanRun := StrAlg.inCanRun;
StrAlg.OpcCommandsDisabled := StrAlg.inOpcCommandsDisabled;

IF StrAlg.isRuning THEN

    StrAlg.hasError := pnsOff.error OR nu1Off.error OR nu2Off.error
    OR stopNU1.error OR stopNU2.error OR testUnsuccessful.error;

    IF puskOilSystem.top THEN
         IF NOT _resetQuestion THEN
         askQuestion(algContinue);
          _resetQuestion:=TRUE;
         END_IF;
    END_IF;

    IF algContinue.answer = _Answers.ANS_YES AND NOT nuOff.top THEN

        runPhase(nuOff);

        IF Im.nu1.onStatus = _statusDualInput.STATUS_ON THEN
		runPhase(nu1Off);
        END_IF;

        IF Im.nu2.onStatus = _statusDualInput.STATUS_ON THEN
		runPhase(nu2Off);
        END_IF;

        resetQuestion(algContinue);

    END_IF;

    IF nuOff.start AND NOT nuOff.top THEN
          runPhase(BreakTest);
	nuOff.top:= Im.nu1.onStatus = _statusDualInput.STATUS_Off
                  AND Im.nu2.onStatus = _statusDualInput.STATUS_Off;
    END_IF;

    IF nuOff.top THEN

        runPhase(dPmgAi);
        runPhase(dPmgDi);
    END_IF;

    (*IF dPmgDi.start AND NOT dPmgDi.top THEN
        dPmgDi.top:=Im.SingleSignals.dP_oilgaz_low.q;
    END_IF;*)

    IF dPmgAi.top AND dPmgDi.top THEN
        runPhase(nuOn);
        runPhase(noRezrv);
    END_IF;

    IF noRezrv.start AND NOT noRezrv.top THEN
        noRezrv.top:=NotHasRezervNU;
    END_IF;

     IF nuOn.start AND (NOT WaitOnNU.Q) THEN
        WaitOnNU(IN:=Im.nu1.onStatus = _statusDualInput.STATUS_On OR
            Im.nu2.onStatus = _statusDualInput.STATUS_On, PT:=T#2S);
        nuOn.top:=Im.nu1.onStatus = _statusDualInput.STATUS_On OR
            Im.nu2.onStatus = _statusDualInput.STATUS_On;
    END_IF;

    IF  WaitOnNU.Q AND noRezrv.top THEN
        ai.Tmasla_MB.Disabled_LA:=TRUE;
        ai.Tmasla_MB.Disabled_LW:=TRUE;
        (*IM.SingleSignals.dP_oilgaz_low.Disabled_Sig:=TRUE;
        IM.SingleSignals.P_oil_low.Disabled_Sig:=TRUE;*)
        ai.Pmasla_posle_GNS.Disabled_LA:=TRUE;
        ai.Pmasla_posle_GNS.Disabled_LW:=TRUE;
        ai.Pmasla_posle_NU.Disabled_LW:=TRUE;

        resetAiProtection(protections.Os_sdvig_nagnetatelja_minus);
        (*resetDiProtection(protections.Vibro_skorost_OP_shesterni_RED_T6);*)
        resetAiProtection(protections.Os_sdvig_nagnetatelja_plus);
        (*resetDiProtection(protections.Vibro_skorost_OP_shesterni_RED_T5);*)

        resetIfRunning(algoritms.autoNu);
        resetIfRunning(algoritms.AutoPns);

        runPhase(stopANU);
        runPhase(pnsOff);

        runPhase(stopNU1);
        runPhase(stopNU2);

    END_IF;

    IF stopANU.start AND NOT stopANU.top THEN

	stopANU.top:= Im.nu1.onStatus = _statusDualInput.STATUS_Off AND
                        Im.nu2.onStatus = _statusDualInput.STATUS_Off;
    END_IF;

    IF BreakTest.top AND NOT pnsOff.top THEN
	testUnsuccessful.error:=TRUE;
    END_IF;

    IF pnsOff.top AND stopANU.top THEN
          resetPhase(BreakTest);
	waitReset(IN:=TRUE, PT:= T#3S);
    END_IF;

    IF waitReset.Q THEN
        algManager.nMode:=ModeGpa.MODE_STOP;
        resetIfRunning(StrAlg);
    END_IF;

    StrAlg.isEnded:= pnsOff.top AND stopANU.top;

END_IF;

StrAlg.CanRun := StrAlg.inCanRun;
StrAlg.OpcCommandsDisabled := StrAlg.inOpcCommandsDisabled;

(* ---- Если управление с ВУ заблокировано, то  передаем команду из алгоритма ---- *)
IF StrAlg.inOpcCommandsDisabled THEN
	StrAlg.inCommand := StrAlg.inCommand_Alg;
ELSE (* иначе передаем команду с АРМа*)
	StrAlg.inCommand := StrAlg.inCommand_ARM;
END_IF;

_sunpackerCommand(command := StrAlg.inCommand);
	source := _sunpackerCommand.source;
	cmd := _sunpackerCommand.cmd;

IF cmd <> 0 AND lastCmd <> cmd AND (((NOT StrAlg.opcCommandsDisabled) AND source > 0) OR source = 0) then
	CASE BYTE_TO_INT(cmd) OF
		(*cmdRun*) 1: 	IF (StrAlg.CanRun) THEN
					StrAlg.isRuning := TRUE;
					StrAlg.isEnded := FALSE;
					StrAlg.hasError := FALSE;
					(*****************       OnRun       *****************)

                                                  algManager.nMode:=ModeGpa.MODE_TESTDPMG;
                                                  resetAndDisable(alg:=algoritms.ppu);
                                                  algoritms.puskOilSystem.inCanRun:= TRUE;
                                                  runPhase(puskOilSystem);

					cmd_for_Status := cmd;
					source_for_Status := source;
					command_error_for_Status := 0;
				ELSE
					StrAlg.isRuning := FALSE;
					StrAlg.isEnded := FALSE;
					StrAlg.hasError 	:= FALSE;

					cmd_for_Status := 0;
					source_for_Status := source;
					command_error_for_Status := cmd;
				END_IF;
		(*cmdReset*) 2: 	StrAlg.isRuning := FALSE;
				StrAlg.isEnded := FALSE;
				StrAlg.hasError 	:= FALSE;

                                         (*****************       OnReset       *****************)
                                        waitReset(IN:=FALSE);
                                        WaitOnNU(IN:=FALSE);
                                        _resetQuestion:=FALSE;
                                        ai.Pmasla_posle_GNS.Disabled_LA:=TRUE;
                                        ai.Pmasla_posle_GNS.Disabled_LW:=TRUE;
                                        ai.Pmasla_posle_NU.Disabled_LW:=TRUE;
                                        (*IM.SingleSignals.P_oil_low.Disabled_Sig:=TRUE;
                                        IM.SingleSignals.dP_oilgaz_low.Disabled_Sig:=TRUE;*)
                                        ai.Tmasla_MB.Disabled_LA:=TRUE;
                                        ai.Tmasla_MB.Disabled_LW:=TRUE;
                                        resetAiProtection(protections.Os_sdvig_nagnetatelja_minus);
                                        (*resetDiProtection(protections.Vibro_skorost_OP_shesterni_RED_T6);*)
                                        resetAiProtection(protections.Os_sdvig_nagnetatelja_plus);
                                        (*resetDiProtection(protections.Vibro_skorost_OP_shesterni_RED_T5);*)

                                        resetPhase(puskOilSystem);
                                        resetPhase(nuOff);
                                        resetPhase(dPmgAi);
                                        resetPhase(dPmgDi);
                                        resetPhase(nuOn);
                                        resetPhase(noRezrv);
                                        resetPhase(BreakTest);
                                        resetPhase(testUnsuccessful);
                                        resetPhase(pnsOff);
                                        resetPhase(stopANU);
                                        resetPhase(nu1Off);
                                        resetPhase(nu2Off);
                                        resetPhase(stopNU1);
                                        resetPhase(stopNU2);

                                        resetQuestion(algContinue);

                                        StrAlg.inOpcCommandsDisabled:=FALSE;

				cmd_for_Status := cmd;
				source_for_Status := source;
				command_error_for_Status := 0;
	END_CASE;
	resetCmdTimer(IN := false);
	resetCmdTimerPriznak := TRUE;
END_IF;
lastCmd := cmd;

resetCmdTimer(IN := resetCmdTimerPriznak, PT := T#5S);
IF resetCmdTimer.Q THEN
	resetCmdTimerPriznak := FALSE;
	source_for_Status := 0;
	cmd_for_Status := 0;
	command_error_for_Status := 0;
END_IF;

StrAlg.Start:= puskOilSystem.startStatus
            OR nuOff.startStatus
            OR dPmgAi.startStatus
            OR dPmgDi.startStatus
            OR nuOn.startStatus
            OR noRezrv.startStatus
            OR BreakTest.startStatus
            OR testUnsuccessful.startStatus
            OR pnsOff.startStatus
            OR stopANU.startStatus
            OR nu1Off.startStatus
            OR nu2Off.startStatus;

StrAlg.Error:=  puskOilSystem.errorStatus
            OR nuOff.errorStatus
            OR dPmgAi.errorStatus
            OR dPmgDi.errorStatus
            OR nuOn.errorStatus
            OR noRezrv.errorStatus
            OR BreakTest.errorStatus
            OR testUnsuccessful.errorStatus
            OR pnsOff.errorStatus
            OR stopANU.errorStatus
            OR nu1Off.errorStatus
            OR nu2Off.errorStatus;

StrAlg.Top:=   puskOilSystem.topStatus
            OR nuOff.topStatus
            OR dPmgAi.topStatus
            OR dPmgDi.topStatus
            OR nuOn.topStatus
            OR noRezrv.topStatus
            OR BreakTest.topStatus
            OR testUnsuccessful.topStatus
            OR pnsOff.topStatus
            OR stopANU.topStatus
            OR nu1Off.topStatus
            OR nu2Off.topStatus;

(*TODO: TYPE PROGRAM CODE HERE*)
StrAlg.status :=  SHL(BYTE_TO_DWORD(source_for_Status), 29)
			OR SHL(BYTE_TO_DWORD(cmd_for_Status), 26)
			OR SHL(BYTE_TO_DWORD(command_error_for_Status), 23)
			OR SHL(BOOL_TO_DWORD(StrAlg.OpcCommandsDisabled ), 21)
			OR SHL(BOOL_TO_DWORD(StrAlg.hasError),4)
			OR SHL(BOOL_TO_DWORD(StrAlg.CanRun),2)
			OR SHL(BOOL_TO_DWORD(StrAlg.isEnded),1)
			OR BOOL_TO_DWORD(StrAlg.isRuning);

(* ---- TestImAlg.st ---- *)
FUNCTION_BLOCK TestImAlg

VAR_IN_OUT
	StrAlg : struct_Alg;
END_VAR

VAR
	_sunpackerCommand : fb_sunpackerCommand;
	source : BYTE;
	cmd : BYTE;
	lastCmd : BYTE;
	source_for_Status : BYTE;
	cmd_for_Status : BYTE;
	command_error_for_Status : BYTE;
	resetCmdTimer : TON;
	resetCmdTimerPriznak : BOOL;
END_VAR

VAR_EXTERNAL
	protectManager : struct_ProtectionsManager;
	algManager : struct_AlgoritmsManager;
	ModeGpa : TYPE_ModeGpa;
	PMcommand : TYPE_CommandsPotectionsManager;
	IM : ImConfig;
END_VAR

StrAlg.CanRun := StrAlg.inCanRun;
StrAlg.OpcCommandsDisabled := StrAlg.inOpcCommandsDisabled;

(* ---- Если управление с ВУ заблокировано, то передаем команду из алгоритма ---- *)
IF StrAlg.inOpcCommandsDisabled THEN
	StrAlg.inCommand := StrAlg.inCommand_Alg;
ELSE (* иначе передаем команду с АРМа*)
	StrAlg.inCommand := StrAlg.inCommand_ARM;
END_IF;

_sunpackerCommand(command := StrAlg.inCommand);
	source := _sunpackerCommand.source;
	cmd := _sunpackerCommand.cmd;

IF cmd <> 0 AND lastCmd <> cmd AND (((NOT StrAlg.opcCommandsDisabled) AND source > 0) OR source = 0) then
	CASE BYTE_TO_INT(cmd) OF
		(*cmdRun*) 1: 	IF (StrAlg.CanRun) THEN
					StrAlg.isRuning := TRUE;
					StrAlg.isEnded := FALSE;
					StrAlg.hasError 	:= FALSE;
                                             (*****************       OnRun       *****************)

                                                      algManager.nMode:=ModeGpa.MODE_TESTIM;
					    UnBlockAllIM(IM);

                                                  (*StrAlg.inOpcCommandsDisabled:=FALSE;*)
					cmd_for_Status := cmd;
					source_for_Status := source;
					command_error_for_Status := 0;
				ELSE
					StrAlg.isRuning := FALSE;
					StrAlg.isEnded := FALSE;
					StrAlg.hasError 	:= FALSE;

					cmd_for_Status := 0;
					source_for_Status := source;
					command_error_for_Status := cmd;
				END_IF;
		(*cmdReset*) 2: 	StrAlg.isRuning := FALSE;
				StrAlg.isEnded := FALSE;
				StrAlg.hasError 	:= FALSE;
                                        (*****************       OnReset       *****************)
                                                  BlockAllIM(IM);
                                                  algManager.nMode:=ModeGpa.MODE_STOP;

				cmd_for_Status := cmd;
				source_for_Status := source;
				command_error_for_Status := 0;
	END_CASE;
	resetCmdTimer(IN := false);
	resetCmdTimerPriznak := TRUE;
END_IF;
lastCmd := cmd;

resetCmdTimer(IN := resetCmdTimerPriznak, PT := T#5S);
IF resetCmdTimer.Q THEN
	resetCmdTimerPriznak := FALSE;
	source_for_Status := 0;
	cmd_for_Status := 0;
	command_error_for_Status := 0;
END_IF;

StrAlg.status :=  SHL(BYTE_TO_DWORD(source_for_Status), 29)
			OR SHL(BYTE_TO_DWORD(cmd_for_Status), 26)
			OR SHL(BYTE_TO_DWORD(command_error_for_Status), 23)
			OR SHL(BOOL_TO_DWORD(StrAlg.OpcCommandsDisabled ), 21)
			OR SHL(BOOL_TO_DWORD(StrAlg.hasError),4)
			OR SHL(BOOL_TO_DWORD(StrAlg.CanRun),2)
			OR SHL(BOOL_TO_DWORD(StrAlg.isEnded),1)
			OR BOOL_TO_DWORD(StrAlg.isRuning);

(* ---- testPmsAlg.st ---- *)
FUNCTION_BLOCK testPmsAlg

VAR_IN_OUT
	StrAlg : struct_Alg;
	algContinue : struct_Question;
END_VAR

VAR
	pnsOn : struct_PhaseAlgoritm;
	PmsUp : struct_PhaseAlgoritm;
	runProtecrionAi : struct_PhaseAlgoritm;
	pnsOff : struct_PhaseAlgoritm;
	BreakTest : struct_PhaseAlgoritm;
	LowOilPS : struct_PhaseAlgoritm;
	LowOilAS : struct_PhaseAlgoritm;
	testUnsuccessful : struct_PhaseAlgoritm;
	fb_pnsOn : fb_ph_Switch;
	fb_PmsUp : fb_ph_WaitAnalogValue;
	fb_algContinue : fb_Question;
	fb_runProtecrionAi : fb_ph_AIprotection;
	fb_pnsOff : fb_ph_Switch;
	fb_BreakTest : fb_ph_Timer;
	fb_LowOilPS : fb_ph_CustomPhase;
	fb_LowOilAS : fb_ph_CustomPhase;
	fb_testUnsuccessful : fb_ph_CustomPhase;
	_sunpackerCommand : fb_sunpackerCommand;
	_DualStateImAction : TYPE_DualStateImAction;
	_Answers : TYPE_Answers;
	_statusDualInput : TYPE_statusDualInput;
	_StatusAi : TYPE_StatusAi;
	_PhaseAlgoritmAction : TYPE_PhaseAlgoritmAction;
	source : BYTE;
	cmd : BYTE;
	lastCmd : BYTE;
	source_for_Status : BYTE;
	cmd_for_Status : BYTE;
	command_error_for_Status : BYTE;
	resetCmdTimer : TON;
	resetCmdTimerPriznak : BOOL;
	onInit : BOOL;
	_resetQuestion : BOOL;
	waitReset : TON;
END_VAR

VAR_EXTERNAL
	IM : ImConfig;
	algoritms : AlgoritmsConfig;
	ai : AiConfig;
	AlgTimers : struct_AlgTimers;
	ModeGpa : TYPE_ModeGpa;
	algManager : struct_AlgoritmsManager;
	protections : ProtectionsConfig;
END_VAR

IF NOT onInit THEN

                   fb_pnsOn(phaseNumber:=0, act:=_on);
        algContinue.AnswerVariants:=_Answers.ANS_YES;
                   fb_PmsUp(phaseNumber:=1);
         fb_runProtecrionAi(phaseNumber:=3, act:=_run);
                  fb_pnsOff(phaseNumber:=4, act:=_off);
               fb_BreakTest(phaseNumber:=5, delay:=T#120S);
                fb_LowOilPS(phaseNumber:=6);
                fb_LowOilAS(phaseNumber:=7);
        fb_testUnsuccessful(phaseNumber:=8);

onInit:=TRUE;
END_IF;

            fb_pnsOn(StrPh:=pnsOn, Im:=IM.pns);
      fb_algContinue(StrQ:=algContinue);
            fb_PmsUp(StrPh:=PmsUp, ai:=ai.Pmasla_posle_GNS, more:=ai.Pmasla_posle_GNS.LW);
  fb_runProtecrionAi(StrPh:=runProtecrionAi, StrAiP:=protections.Os_sdvig_nagnetatelja_minus);
           fb_pnsOff(StrPh:=pnsOff, Im:=IM.pns);
        fb_BreakTest(StrPh:=BreakTest, timer:=AlgTimers.testPms_BreakTest);
         fb_LowOilPS(StrPh:=LowOilPS);
         fb_LowOilAS(StrPh:=LowOilAS);
 fb_testUnsuccessful(StrPh:=testUnsuccessful);

StrAlg.CanRun := StrAlg.inCanRun;
StrAlg.OpcCommandsDisabled := StrAlg.inOpcCommandsDisabled;

IF StrAlg.isRuning THEN

    StrAlg.hasError := pnsOn.error OR pnsOff.error OR testUnsuccessful.error;

    IF pnsOn.top THEN
         runPhase(PmsUp);
    END_IF;

    IF PmsUp.top THEN
         runPhase(runProtecrionAi);
    END_IF;

    IF runProtecrionAi.top THEN
         (*IM.SingleSignals.P_oil_low.Disabled_Sig:=FALSE;*)
         ai.Pmasla_posle_GNS.Disabled_LA:=FALSE;
         ai.Pmasla_posle_GNS.Disabled_LW:=FALSE;
         ai.Pmasla_posle_NU.Disabled_LW:=FALSE;
             IF NOT _resetQuestion THEN
                 askQuestion(algContinue);
                 _resetQuestion:=TRUE;
             END_IF;
    END_IF;

    IF algContinue.answer = _Answers.ANS_YES THEN

        runPhase(BreakTest);
        runPhase(pnsOff);
        runPhase(LowOilPS);
        runPhase(LowOilAS);
        resetQuestion(algContinue);

    END_IF;

    IF 	LowOilPS.start AND NOT LowOilPS.top THEN
	LowOilPS.top:= ai.Pmasla_posle_GNS.interval = _statusAi.LW;
    END_IF;
    IF 	LowOilAS.start AND NOT LowOilAS.top THEN
	LowOilAS.top:= ai.Pmasla_posle_GNS.interval = _statusAi.LA;
    END_IF;

    IF LowOilPS.top AND LowOilAS.top THEN
          resetPhase(BreakTest);
          waitReset(IN:=TRUE, PT:= T#3S);
    END_IF;

    IF BreakTest.top AND StrAlg.isEnded THEN
	testUnsuccessful.error:=TRUE;
    END_IF;

    IF waitReset.Q THEN
        algManager.nMode:=ModeGpa.MODE_STOP;
        resetIfRunning(StrAlg);
    END_IF;

    StrAlg.isEnded:= LowOilPS.top AND LowOilAS.top;

END_IF;

StrAlg.CanRun := StrAlg.inCanRun;
StrAlg.OpcCommandsDisabled := StrAlg.inOpcCommandsDisabled;

(* ---- Если управление с ВУ заблокировано, то  передаем команду из алгоритма ---- *)
IF StrAlg.inOpcCommandsDisabled THEN
	StrAlg.inCommand := StrAlg.inCommand_Alg;
ELSE (* иначе передаем команду с АРМа*)
	StrAlg.inCommand := StrAlg.inCommand_ARM;
END_IF;

_sunpackerCommand(command := StrAlg.inCommand);
	source := _sunpackerCommand.source;
	cmd := _sunpackerCommand.cmd;

IF cmd <> 0 AND lastCmd <> cmd AND (((NOT StrAlg.opcCommandsDisabled) AND source > 0) OR source = 0) then
	CASE BYTE_TO_INT(cmd) OF
		(*cmdRun*) 1: 	IF (StrAlg.CanRun) THEN
					StrAlg.isRuning := TRUE;
					StrAlg.isEnded := FALSE;
					StrAlg.hasError := FALSE;
					(*****************       OnRun       *****************)

                                                  algManager.nMode:=ModeGpa.MODE_TESTPMS;
                                                  resetAndDisable(alg:=algoritms.ppu);
                                                  runPhase(pnsOn);

					cmd_for_Status := cmd;
					source_for_Status := source;
					command_error_for_Status := 0;
				ELSE
					StrAlg.isRuning := FALSE;
					StrAlg.isEnded := FALSE;
					StrAlg.hasError 	:= FALSE;

					cmd_for_Status := 0;
					source_for_Status := source;
					command_error_for_Status := cmd;
				END_IF;
		(*cmdReset*) 2: 	StrAlg.isRuning := FALSE;
				StrAlg.isEnded := FALSE;
				StrAlg.hasError 	:= FALSE;

                                         (*****************       OnReset       *****************)
                                        waitReset(IN:=FALSE);
                                        _resetQuestion:=FALSE;
                                        ai.Pmasla_posle_GNS.Disabled_LA:=TRUE;
                                        ai.Pmasla_posle_GNS.Disabled_LW:=TRUE;
                                        ai.Pmasla_posle_NU.Disabled_LW:=TRUE;
                                       (* IM.SingleSignals.P_oil_low.Disabled_Sig:=TRUE;*)
                                        resetAiProtection(protections.Os_sdvig_nagnetatelja_minus);

                                        resetPhase(pnsOn);
                                        resetPhase(PmsUp);
                                        resetPhase(runProtecrionAi);
                                        resetPhase(pnsOff);
                                        resetPhase(BreakTest);
                                        resetPhase(LowOilPS);
                                        resetPhase(LowOilAS);
                                        resetPhase(testUnsuccessful);

                                        resetQuestion(algContinue);

                                        StrAlg.inOpcCommandsDisabled:=FALSE;

				cmd_for_Status := cmd;
				source_for_Status := source;
				command_error_for_Status := 0;
	END_CASE;
	resetCmdTimer(IN := false);
	resetCmdTimerPriznak := TRUE;
END_IF;
lastCmd := cmd;

resetCmdTimer(IN := resetCmdTimerPriznak, PT := T#5S);
IF resetCmdTimer.Q THEN
	resetCmdTimerPriznak := FALSE;
	source_for_Status := 0;
	cmd_for_Status := 0;
	command_error_for_Status := 0;
END_IF;

StrAlg.Start:= pnsOn.startStatus
            OR PmsUp.startStatus
            OR runProtecrionAi.startStatus
            OR pnsOff.startStatus
            OR BreakTest.startStatus
            OR LowOilPS.startStatus
            OR LowOilAS.startStatus
            OR testUnsuccessful.startStatus;

StrAlg.Error:= pnsOn.errorStatus
            OR PmsUp.errorStatus
            OR runProtecrionAi.errorStatus
            OR pnsOff.errorStatus
            OR BreakTest.errorStatus
            OR LowOilPS.errorStatus
            OR LowOilAS.errorStatus
            OR testUnsuccessful.errorStatus;

StrAlg.Top:=   pnsOn.topStatus
            OR PmsUp.topStatus
            OR runProtecrionAi.topStatus
            OR pnsOff.topStatus
            OR BreakTest.topStatus
            OR LowOilPS.topStatus
            OR LowOilAS.topStatus
            OR testUnsuccessful.topStatus;

(*TODO: TYPE PROGRAM CODE HERE*)
StrAlg.status :=  SHL(BYTE_TO_DWORD(source_for_Status), 29)
			OR SHL(BYTE_TO_DWORD(cmd_for_Status), 26)
			OR SHL(BYTE_TO_DWORD(command_error_for_Status), 23)
			OR SHL(BOOL_TO_DWORD(StrAlg.OpcCommandsDisabled ), 21)
			OR SHL(BOOL_TO_DWORD(StrAlg.hasError),4)
			OR SHL(BOOL_TO_DWORD(StrAlg.CanRun),2)
			OR SHL(BOOL_TO_DWORD(StrAlg.isEnded),1)
			OR BOOL_TO_DWORD(StrAlg.isRuning);

(* ---- TestProtectionAlg.st ---- *)
FUNCTION_BLOCK TestProtectionAlg

VAR_IN_OUT
	StrAlg : struct_Alg;
END_VAR

VAR
	_sunpackerCommand : fb_sunpackerCommand;
	source : BYTE;
	cmd : BYTE;
	lastCmd : BYTE;
	source_for_Status : BYTE;
	cmd_for_Status : BYTE;
	command_error_for_Status : BYTE;
	resetCmdTimer : TON;
	resetCmdTimerPriznak : BOOL;
END_VAR

VAR_EXTERNAL
	ai : AiConfig;
	protectManager : struct_ProtectionsManager;
	algManager : struct_AlgoritmsManager;
	ModeGpa : TYPE_ModeGpa;
	PMcommand : TYPE_CommandsPotectionsManager;
	IM : ImConfig;
END_VAR

StrAlg.CanRun := StrAlg.inCanRun;
StrAlg.OpcCommandsDisabled := StrAlg.inOpcCommandsDisabled;

(* ---- Если управление с ВУ заблокировано, то передаем команду из алгоритма ---- *)
IF StrAlg.inOpcCommandsDisabled THEN
	StrAlg.inCommand := StrAlg.inCommand_Alg;
ELSE (* иначе передаем команду с АРМа*)
	StrAlg.inCommand := StrAlg.inCommand_ARM;
END_IF;

_sunpackerCommand(command := StrAlg.inCommand);
	source := _sunpackerCommand.source;
	cmd := _sunpackerCommand.cmd;

IF cmd <> 0 AND lastCmd <> cmd AND (((NOT StrAlg.opcCommandsDisabled) AND source > 0) OR source = 0) then
	CASE BYTE_TO_INT(cmd) OF
		(*cmdRun*) 1: 	IF (StrAlg.CanRun) THEN
					StrAlg.isRuning := TRUE;
					StrAlg.isEnded := FALSE;
					StrAlg.hasError 	:= FALSE;
                                             (*****************       OnRun       *****************)
                                                      algManager.nMode:=ModeGpa.MODE_TESTAZ;
                                                      protectManager.inCommand:=PMcommand.CheckProtections;
					    EnableAiLimits(ai);
                                                      (*IM.SingleSignals.P_oil_low.Disabled_Sig:=FALSE;*)
                                                      (*IM.SingleSignals.dP_oilgaz_low.Disabled_Sig:=FALSE;*)
                                                  (*StrAlg.inOpcCommandsDisabled:=FALSE;*)
					cmd_for_Status := cmd;
					source_for_Status := source;
					command_error_for_Status := 0;
				ELSE
					StrAlg.isRuning := FALSE;
					StrAlg.isEnded := FALSE;
					StrAlg.hasError 	:= FALSE;

					cmd_for_Status := 0;
					source_for_Status := source;
					command_error_for_Status := cmd;
				END_IF;
		(*cmdReset*) 2: 	StrAlg.isRuning := FALSE;
				StrAlg.isEnded := FALSE;
				StrAlg.hasError 	:= FALSE;
                                        (*****************       OnReset       *****************)
                                                  DisableAiLimits(ai);
                                                  (*IM.SingleSignals.P_oil_low.Disabled_Sig:=TRUE;
                                                  IM.SingleSignals.dP_oilgaz_low.Disabled_Sig:=TRUE;*)
                                                  protectManager.inCommand:=PMcommand.RestartAllProtections;
                                                  algManager.nMode:=ModeGpa.MODE_STOP;

				cmd_for_Status := cmd;
				source_for_Status := source;
				command_error_for_Status := 0;
	END_CASE;
	resetCmdTimer(IN := false);
	resetCmdTimerPriznak := TRUE;
END_IF;
lastCmd := cmd;

resetCmdTimer(IN := resetCmdTimerPriznak, PT := T#5S);
IF resetCmdTimer.Q THEN
	resetCmdTimerPriznak := FALSE;
	source_for_Status := 0;
	cmd_for_Status := 0;
	command_error_for_Status := 0;
END_IF;

StrAlg.status :=  SHL(BYTE_TO_DWORD(source_for_Status), 29)
			OR SHL(BYTE_TO_DWORD(cmd_for_Status), 26)
			OR SHL(BYTE_TO_DWORD(command_error_for_Status), 23)
			OR SHL(BOOL_TO_DWORD(StrAlg.OpcCommandsDisabled ), 21)
			OR SHL(BOOL_TO_DWORD(StrAlg.hasError),4)
			OR SHL(BOOL_TO_DWORD(StrAlg.CanRun),2)
			OR SHL(BOOL_TO_DWORD(StrAlg.isEnded),1)
			OR BOOL_TO_DWORD(StrAlg.isRuning);
